// TIA Portal project "Phase_Two" (V15.1)

(* hardware
DEVICE "S71500/ET200MP-Station_1"  S7-1500 station
   slot 0: "Profilschiene_0"  6ES7 590-1***0-0AA0
   slot 1: "PLC_1"  CPU 1511-1 PN  6ES7 511-1AK00-0AB0  V1.8
   slot 2: "AI 8xU/I/RTD/TC ST_1"  AI 8xU/I/RTD/TC ST  6ES7 531-7KF00-0AB0  V2.0
   slot 3: "AI 8xU/I/RTD/TC ST_2"  AI 8xU/I/RTD/TC ST  6ES7 531-7KF00-0AB0  V2.0
   slot 4: "AI 8xU/I/RTD/TC ST_3"  AI 8xU/I/RTD/TC ST  6ES7 531-7KF00-0AB0  V2.0
   slot 5: "AI 8xU/I/RTD/TC ST_4"  AI 8xU/I/RTD/TC ST  6ES7 531-7KF00-0AB0  V2.0
   slot 6: "DI 16x24VDC BA_1"  DI 16x24VDC BA  6ES7 521-1BH10-0AA0  V1.0
   slot 7: "AI 8xU/I/RTD/TC ST_5"  AI 8xU/I/RTD/TC ST  6ES7 531-7KF00-0AB0  V2.0
DEVICE "HMI_2"  TP1200 Comfort
   slot 0: "HMI_2"  TP1200 Comfort  6AV2 124-0MC01-0AX0  15.1.0.0
   slot 1: "HMI_RT_2"  TP1200 Comfort  6AV2 124-0MC01-0AX0  15.1.0.0
   slot 5: "HMI_2.IE_CP_1"  PROFINET Interface  15.0.1.0
      slot 1: "PROFINET Interface_1"  PROFINET Interface
         slot 1: "Port_1"  Port
         slot 2: "Port_2"  Port
   slot 7: "HMI_2.MPI/DP_CP_1"  MPI/DP Interface  15.0.1.0
*)

// ===== PLC "PLC_1"  CPU 1511-1 PN =====

VAR_GLOBAL   // PLC tag table "Standard-Variablentabelle"
   "Item at entry" AT %E0.0 : Bool;
   "Item at Exit" AT %I0.1 : Bool;
   "Moving x" AT %I0.2 : Bool;
   "Item Detected" AT %I0.4 : Bool;
   "Start" AT %I0.5 : Bool;
   "Reset" AT %I0.6 : Bool;
   "Stop" AT %I0.7 : Bool;
   "Entry Conveyor" AT %QW6 : Word;
   "Exit Conveyor" AT %QW8 : Word;
   "Move x" AT %QW18 : Word;
   "Move z" AT %QW20 : Word;
   "Grab" AT %Q0.4 : Bool;
   "Start Light" AT %Q0.5 : Bool;
   "Reset Light" AT %Q0.6 : Bool;
   "Stop Light" AT %Q0.7 : Bool;
   "Moving Z" AT %I0.3 : Bool;
   "-ve edge z" AT %M7.0 : Bool;
   "Emergency Stop" AT %I1.0 : Bool;
   "-ve edge x" AT %M7.1 : Bool;
   "-ve edge to start z" AT %M7.2 : Bool;
   "-ve edge to start x" AT %M7.3 : Bool;
   "o/ps off" AT %M7.4 : Bool;
   "stop tag" AT %M7.5 : Bool;
   "Entry_conv_true" AT %M0.0 : Bool;
   "Norm_Entry_conv" AT %MD100 : Real;
   "Exit_Conv_true" AT %M0.1 : Bool;
   "Norm_Exit_conv" AT %MD104 : Real;
   "Feeding_Curved_Conv" AT %QW10 : Word;
   "Norm_Feeding_Curved_Conv" AT %MD108 : Real;
   "To Sorting Conv" AT %QW12 : Word;
   "Blue Conv" AT %QW14 : Word;
   "Green Conv" AT %QW16 : Word;
   "Sorting Rollers" AT %Q1.0 : Bool;
   "Right Pose" AT %Q1.1 : Bool;
   "Left Pose" AT %Q1.2 : Bool;
   "Vision Sensor Blue" AT %I1.3 : Bool;
   "Vision Sensor Green" AT %I1.4 : Bool;
   "Move_x_True" AT %M0.2 : Bool;
   "Move_z_True" AT %M0.3 : Bool;
   "Moving_x_Normalized" AT %M0.4 : Bool;
   "Moving_z_Normalized" AT %M0.5 : Bool;
   "Norm_Move_x" AT %MD112 : Real;
   "Norm _Move z" AT %MD116 : Real;
   "Start Green Conv sesnor" AT %I1.5 : Bool;
   "Start Blue Conv sensor" AT %I1.6 : Bool;
   "Start Green conv bit" AT %M0.6 : Bool;
   "Start Blue Conv bit" AT %M0.7 : Bool;
   "Green Machining Sensor Exit" AT %I2.0 : Bool;
   "Blue Machining Sensor Exit" AT %I1.7 : Bool;
   "Blue Conv 2" AT %QW22 : Word;
   "Green Conv 2" AT %QW24 : Word;
   "Green Conv 3" AT %QW26 : Word;
   "Green Conv 4" AT %QW28 : Word;
   "Machining Blue Start" AT %Q1.3 : Bool;
   "Machining Blue prod_lid" AT %Q1.4 : Bool;
   "-ve edge to start b_machining" AT %M10.0 : Bool;
   "Start b_machining bit" AT %M10.1 : Bool;
   "-ve edge to start g_machining" AT %M10.2 : Bool;
   "Start g_machining bit" AT %M10.3 : Bool;
   "Machining Green Start" AT %Q1.5 : Bool;
   "Machining Green prod_lid" AT %Q1.6 : Bool;
   "Green Conv after mach." AT %QW30 : Word;
   "Blue Conv after mach." AT %QW32 : Word;
   "Green Conv to Assembly" AT %QW34 : Word;
   "Curvred Green Conv assembly" AT %QW36 : Word;
   "Green lid Conv Assembly" AT %QW38 : Word;
   "Green Base Conv Assembly" AT %QW40 : Word;
   "Move_x Green Asssembly" AT %QW42 : Word;
   "Move_z Green Assembly" AT %QW44 : Word;
   "Moving_x Green Assembly" AT %I2.1 : Bool;
   "Moving_z Green Assembly" AT %I2.2 : Bool;
   "Item Detected Green Assembly" AT %I2.3 : Bool;
   "Grab Green Assembly" AT %Q1.7 : Bool;
   "Green Base Assembly Sensor" AT %I2.4 : Bool;
   "Green Lid Assembly Sensor" AT %I2.5 : Bool;
   "Green Base Vision Sensor" AT %I2.6 : Bool;
   "Pusher Green Base" AT %Q2.0 : Bool;
   "Pusher Green F_Limit" AT %I2.7 : Bool;
   "+ve edge Pusher Green" AT %M12.0 : Bool;
   "+ve edge Pusher Green true" AT %M12.1 : Bool;
   "Green Lid Vision Sensor" AT %I3.0 : Bool;
   "+ve edge green base sesnsor" AT %M15.0 : Bool;
   "+ve edge green lid sensor" AT %M15.1 : Bool;
   "Clamp Green Lid" AT %Q2.1 : Bool;
   "Clamp Green Base" AT %Q2.2 : Bool;
   "Green Base Clamped" AT %I3.2 : Bool;
   "Green Lid Clamped" AT %I3.1 : Bool;
   "Green Product Raise" AT %Q2.3 : Bool;
   "Green Product Base Limit" AT %I3.3 : Bool;
   "+ve edge to release clamp ( Green base)" AT %M20.0 : Bool;
   "+ve edge to release G Base true" AT %M20.1 : Bool;
   "Tag_1" AT %M50.0 : Bool;
   "Tag_2" AT %M25.0 : Bool;
   "Tag_3" AT %M60.0 : Bool;
   "Tag_4" AT %M61.0 : Bool;
   "+ve edge to release G lid (true)" AT %M61.1 : Bool;
   "Tag_5" AT %M65.0 : Bool;
   "Tag_6" AT %M80.0 : Bool;
   "Move z True green" AT %M80.1 : Bool;
   "move x True green" AT %M80.2 : Bool;
   "Tag_7" AT %M30.0 : Bool;
   "Tag_8" AT %M30.1 : Bool;
   "-ve edge to start x green" AT %M30.2 : Bool;
   "Move_x Green True" AT %M30.3 : Bool;
   "Tag_9" AT %M150.0 : Bool;
   "-ve edge to start z green" AT %M150.1 : Bool;
   "o/ps off green" AT %M200.0 : Bool;
   "Tag_10" AT %M210.0 : Bool;
   "Tag_11" AT %M55.0 : Bool;
   "FreeBase" AT %M30.4 : Bool;
   "Tag_12" AT %M40.0 : Bool;
   "Tag_13" AT %M40.1 : Bool;
   "Tag_14" AT %M40.3 : Bool;
   "Tag_15" AT %M40.2 : Bool;
   "Tag_16" AT %M40.4 : Bool;
   "Tag_17" AT %M40.5 : Bool;
   "Tag_18" AT %M40.6 : Bool;
   "Tag_19" AT %M40.7 : Bool;
   "Tag_20" AT %M41.0 : Bool;
   "GreenPositionerRaise" AT %Q2.4 : Bool;
   "Tag_21" AT %M41.2 : Bool;
   "Tag_22" AT %M41.3 : Bool;
   "Tag_23" AT %M41.4 : Bool;
   "Tag_24" AT %M41.5 : Bool;
   "Tag_25" AT %M41.6 : Bool;
   "Blue Base Assembly Sensor" AT %I3.7 : Bool;
   "Blue Lid Assembly Sensor" AT %I4.0 : Bool;
   "Blue Base Clamped" AT %I4.1 : Bool;
   "Blue Lid Clamped" AT %I4.2 : Bool;
   "Blue Product Counter Sensor" AT %I4.3 : Bool;
   "Blue Pusher Front Limit" AT %I4.4 : Bool;
   "Item Detected Blue" AT %I3.6 : Bool;
   "Grab Blue" AT %Q2.5 : Bool;
   "Blue Base Clamp" AT %Q2.6 : Bool;
   "Blue lid Clamp" AT %Q2.7 : Bool;
   "Blue Base Freed" AT %Q3.0 : Bool;
   "Blue lid Freed" AT %Q3.1 : Bool;
   "Pusher Blue Base" AT %Q3.2 : Bool;
   "Vision Sensor Blue base" AT %IW5 : Word;
   "Move_X Blue" AT %QW46 : Word;
   "Move_Z Blue" AT %QW48 : Word;
   "Blue Base Conv Assembly" AT %QW50 : Word;
   "Curved Blue Lid Conv Assembly" AT %QW52 : Word;
   "Blue Lid Conv Assembly" AT %QW54 : Word;
   "Moving_X Blue" AT %I4.5 : Bool;
   "Moving_Z Blue" AT %I4.6 : Bool;
   "Blue Base sensor" AT %M300.0 : Bool;
   "+ve edge Pusher blue true" AT %M300.1 : Bool;
   "Tag_26" AT %M300.2 : Bool;
   "Tag_27" AT %M300.3 : Bool;
   "Blue Lid Sensor" AT %M300.4 : Bool;
   "Tag_28" AT %M300.5 : Bool;
   "Tag_29" AT %M300.6 : Bool;
   "Tag_30" AT %M300.7 : Bool;
   "-ve edge to start Z blue" AT %M301.0 : Bool;
   "Free base blue" AT %M301.1 : Bool;
   "Tag_31" AT %M301.2 : Bool;
   "Tag_32" AT %M301.3 : Bool;
   "+ve edge to relase  b lid (true)" AT %M301.4 : Bool;
   "Tag_33" AT %M301.5 : Bool;
   "Tag_34" AT %M301.6 : Bool;
   "Move z true Blue" AT %M301.7 : Bool;
   "Tag_35" AT %M302.0 : Bool;
   "Tag_36" AT %M5.0 : Bool;
   "Tag_37" AT %M302.2 : Bool;
   "Tag_38" AT %M500.1 : Bool;
   "Tag_39" AT %M302.4 : Bool;
   "-ve edge to start X blue" AT %M302.5 : Bool;
   "Tag_40" AT %M302.6 : Bool;
   "Move_x Blue True" AT %M302.7 : Bool;
   "Tag_41" AT %M303.0 : Bool;
   "Tag_42" AT %M303.1 : Bool;
   "Tag_43" AT %M303.2 : Bool;
   "Blue Product Base Limit" AT %I3.5 : Bool;
   "Tag_44" AT %M303.4 : Bool;
   "Tag_45" AT %M303.5 : Bool;
   "Tag_46" AT %M303.6 : Bool;
   "Tag_47" AT %M303.7 : Bool;
   "Tag_48" AT %M304.0 : Bool;
   "Tag_49" AT %M304.1 : Bool;
   "Tag_50" AT %M500.2 : Bool;
   "Tag_51" AT %M600.0 : Bool;
   "tag_52" AT %M600.1 : Bool;
   "Tag_53" AT %M600.2 : Bool;
   "Tag_54" AT %M600.3 : Bool;
   "RequiredGreen" AT %MW700 : Word;
   "RequiredBlue" AT %MW702 : Word;
   "DoubleRequiredBlue" AT %MW704 : Word;
   "DoubleRequiredGreen" AT %MW706 : Word;
   "ReachedBlueItems" AT %M600.4 : Bool;
   "ReachedGreenItems" AT %M600.5 : Bool;
   "GreenProductCounterSensor" AT %I3.4 : Bool;
   "DoneGreen" AT %MW708 : Word;
   "DoneBlue" AT %MW710 : Word;
   "RequiredBlue+1" AT %MW712 : Word;
   "RequiredGreen+1" AT %MW714 : Word;
   "Reset_Tag" AT %M600.6 : Bool;
   "DoubleRequiredBlue+1" AT %MW716 : Word;
   "DoubleRequiredGreen+1" AT %MW718 : Word;
   "InputConvOFF" AT %M600.7 : Bool;
   "ReachedRawGreen" AT %M601.0 : Bool;
   "ReachedRawBlue" AT %M601.1 : Bool;
   "ConvSpeedBeforeMach" AT %MW720 : Word;
   "ConvSpeedAfterMach" AT %MW722 : Word;
   "StopConvBM" AT %M601.2 : Bool;
   "Reset_Tag_2" AT %M601.3 : Bool;
   "StartFromHmi" AT %M601.4 : Bool;
   "StopFromHmi" AT %M601.5 : Bool;
   "ResetFromHmi" AT %M601.6 : Bool;
   "Conv_Speed_Before_mach_Hmi" AT %MW724 : Word;
   "Conv_Speed_after_mach_Hmi" AT %MW726 : Word;
   "Normalized Conv Before mach" AT %MD120 : Real;
   "Normalized Conv After mach" AT %MD124 : Real;
END_VAR

// folder: System blocks/Program resources

DATA_BLOCK "IEC_Timer_0_DB"   // DB1
{ S7_Optimized_Access := 'TRUE' }
AUTHOR : Simatic
FAMILY : IEC
NAME : IEC_TMR
VERSION : 1.0
// stored: InstanceOfName IEC_TIMER
"IEC_TIMER"
BEGIN
END_DATA_BLOCK

DATA_BLOCK "IEC_Counter_0_DB"   // DB3
{ S7_Optimized_Access := 'TRUE' }
AUTHOR : Simatic
FAMILY : IEC
NAME : CNTR
VERSION : 1.0
// stored: InstanceOfName IEC_COUNTER
"IEC_COUNTER"
BEGIN
END_DATA_BLOCK

DATA_BLOCK "IEC_Counter_0_DB_1"   // DB4
{ S7_Optimized_Access := 'TRUE' }
AUTHOR : Simatic
FAMILY : IEC
NAME : CNTR
VERSION : 1.0
// stored: InstanceOfName IEC_COUNTER
"IEC_COUNTER"
BEGIN
END_DATA_BLOCK

DATA_BLOCK "IEC_Counter_0_DB_2"   // DB5
{ S7_Optimized_Access := 'TRUE' }
AUTHOR : Simatic
FAMILY : IEC
NAME : CNTR
VERSION : 1.0
// stored: InstanceOfName IEC_COUNTER
"IEC_COUNTER"
BEGIN
END_DATA_BLOCK

DATA_BLOCK "IEC_Counter_0_DB_3"   // DB6
{ S7_Optimized_Access := 'TRUE' }
AUTHOR : Simatic
FAMILY : IEC
NAME : CNTR
VERSION : 1.0
// stored: InstanceOfName IEC_COUNTER
"IEC_COUNTER"
BEGIN
END_DATA_BLOCK

DATA_BLOCK "IEC_Counter_0_DB_4"   // DB7
{ S7_Optimized_Access := 'TRUE' }
AUTHOR : Simatic
FAMILY : IEC
NAME : CNTR
VERSION : 1.0
// stored: InstanceOfName IEC_COUNTER
"IEC_COUNTER"
BEGIN
END_DATA_BLOCK

DATA_BLOCK "IEC_Timer_0_DB_4"   // DB8
{ S7_Optimized_Access := 'TRUE' }
AUTHOR : Simatic
FAMILY : IEC
NAME : IEC_TMR
VERSION : 1.0
// stored: InstanceOfName IEC_TIMER
"IEC_TIMER"
BEGIN
END_DATA_BLOCK

DATA_BLOCK "IEC_Timer_0_DB_5"   // DB9
{ S7_Optimized_Access := 'TRUE' }
AUTHOR : Simatic
FAMILY : IEC
NAME : IEC_TMR
VERSION : 1.0
// stored: InstanceOfName IEC_TIMER
"IEC_TIMER"
BEGIN
END_DATA_BLOCK

DATA_BLOCK "IEC_Timer_0_DB_6"   // DB10
{ S7_Optimized_Access := 'TRUE' }
AUTHOR : Simatic
FAMILY : IEC
NAME : IEC_TMR
VERSION : 1.0
// stored: InstanceOfName IEC_TIMER
"IEC_TIMER"
BEGIN
END_DATA_BLOCK

DATA_BLOCK "IEC_Timer_0_DB_7"   // DB11
{ S7_Optimized_Access := 'TRUE' }
AUTHOR : Simatic
FAMILY : IEC
NAME : IEC_TMR
VERSION : 1.0
// stored: InstanceOfName IEC_TIMER
"IEC_TIMER"
BEGIN
END_DATA_BLOCK

DATA_BLOCK "IEC_Counter_0_DB_5"   // DB12
{ S7_Optimized_Access := 'TRUE' }
AUTHOR : Simatic
FAMILY : IEC
NAME : CNTR
VERSION : 1.0
// stored: InstanceOfName IEC_COUNTER
"IEC_COUNTER"
BEGIN
END_DATA_BLOCK

DATA_BLOCK "IEC_Counter_0_DB_6"   // DB13
{ S7_Optimized_Access := 'TRUE' }
AUTHOR : Simatic
FAMILY : IEC
NAME : CNTR
VERSION : 1.0
// stored: InstanceOfName IEC_COUNTER
"IEC_COUNTER"
BEGIN
END_DATA_BLOCK

DATA_BLOCK "IEC_Timer_0_DB_2"   // DB14
{ S7_Optimized_Access := 'TRUE' }
AUTHOR : Simatic
FAMILY : IEC
NAME : IEC_TMR
VERSION : 1.0
// stored: InstanceOfName IEC_TIMER
"IEC_TIMER"
BEGIN
END_DATA_BLOCK

DATA_BLOCK "IEC_Timer_0_DB_3"   // DB15
{ S7_Optimized_Access := 'TRUE' }
AUTHOR : Simatic
FAMILY : IEC
NAME : IEC_TMR
VERSION : 1.0
// stored: InstanceOfName IEC_TIMER
"IEC_TIMER"
BEGIN
END_DATA_BLOCK

// folder: (top level)

FUNCTION "MHJ-PLC-Lab-Function-S71500" : Void   // FC9000, SCL
{ S7_Optimized_Access := 'TRUE' }
VERSION : 0.1
   VAR_TEMP
      Value : Byte;
      ForCounter : Int;
   END_VAR
   VAR CONSTANT
      Value_01_DW : DWord := 16#1223_5486;
      Value_02_DW : DWord := 16#A6C9_D1F5;
   END_VAR
BEGIN

   #Value:=PEEK(area := 16#82,
        dbNumber := 0,
        byteOffset := 511);
   #Value := #Value + 1;

   POKE(area := 16#82,
        dbNumber := 0,
        byteOffset := 511,
        value := #Value);

   POKE(area := 16#82,
        dbNumber := 0,
        byteOffset := 1016,
        value := #Value_01_DW);
   POKE(area := 16#82,
        dbNumber := 0,
        byteOffset := 1020,
        value := #Value_02_DW);

   FOR #ForCounter := 0 TO 63 DO
       #Value:=PEEK(area := 16#1,
            dbNumber := 0,
            byteOffset := #ForCounter);
       POKE(area := 16#81,
            dbNumber := 0,
            byteOffset := #ForCounter,
            value := #Value);
   END_FOR;
   #Value := PEEK(area := 16#1,
                  dbNumber := 0,
                  byteOffset := 512);
   POKE(area := 16#82,
        dbNumber := 0,
        byteOffset := 512,
        value := #Value);
END_FUNCTION

ORGANIZATION_BLOCK "Main"   // OB1, FBD, ProgramCycle
TITLE = "Main Program Sweep (Cycle)"
{ S7_Optimized_Access := 'TRUE' }
VERSION : 0.1
   VAR_INPUT
      Initial_Call : Bool;   // Initial call of this OB
      Remanence : Bool;   // =True, if remanent data are available
   END_VAR
BEGIN

REGION Network 1
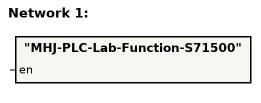
   "MHJ-PLC-Lab-Function-S71500"();
END_REGION
END_ORGANIZATION_BLOCK

ORGANIZATION_BLOCK "Main_1"   // OB123, LAD, ProgramCycle
TITLE = "Main Program Sweep (Cycle)"
{ S7_Optimized_Access := 'TRUE' }
VERSION : 0.1
   VAR_INPUT
      Initial_Call : Bool;   // Initial call of this OB
      Remanence : Bool;   // =True, if remanent data are available
   END_VAR
   VAR_TEMP   // added for the SCL form of the ladder/FBD networks
      _w1 : Bool;
      _w2 : Bool;
      _w3 : Bool;
      _w4 : Bool;
   END_VAR
BEGIN

REGION Network 1
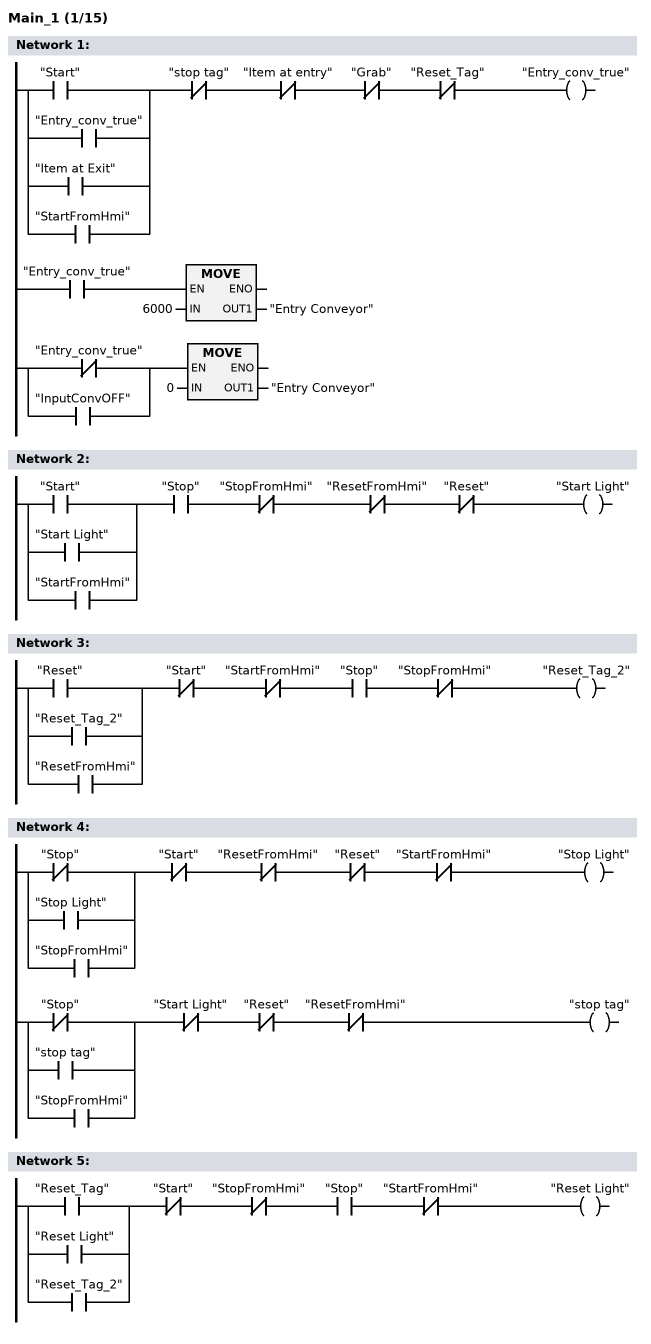
   RUNG wire#powerrail
      Contact( "Start" )
      wire#w1
      I_Contact( "stop tag" )
      I_Contact( "Item at entry" )
      I_Contact( "Grab" )
      I_Contact( "Reset_Tag" )
      Coil( "Entry_conv_true" )
   END_RUNG
   RUNG wire#powerrail
      Contact( "Entry_conv_true" )
   END_RUNG wire#w1
   RUNG wire#powerrail
      Contact( "Item at Exit" )
   END_RUNG wire#w1
   RUNG wire#powerrail
      Contact( "StartFromHmi" )
   END_RUNG wire#w1
   RUNG wire#powerrail
      Contact( "Entry_conv_true" )
      Move(in := 6000, out1 => "Entry Conveyor")
   END_RUNG
   RUNG wire#powerrail
      I_Contact( "Entry_conv_true" )
      wire#w2
      Move(in := 0, out1 => "Entry Conveyor")
   END_RUNG
   RUNG wire#powerrail
      Contact( "InputConvOFF" )
   END_RUNG wire#w2
   // the same network as SCL:
   "Entry_conv_true" := ("Start" OR "Entry_conv_true" OR "Item at Exit" OR "StartFromHmi") AND NOT "stop tag" AND NOT "Item at entry" AND NOT "Grab" AND NOT "Reset_Tag";
   IF "Entry_conv_true" THEN "Entry Conveyor" := 6000; END_IF;
   IF NOT "Entry_conv_true" OR "InputConvOFF" THEN "Entry Conveyor" := 0; END_IF;
END_REGION

REGION Network 2
   RUNG wire#powerrail
      Contact( "Start" )
      wire#w1
      Contact( "Stop" )
      I_Contact( "StopFromHmi" )
      I_Contact( "ResetFromHmi" )
      I_Contact( "Reset" )
      Coil( "Start Light" )
   END_RUNG
   RUNG wire#powerrail
      Contact( "Start Light" )
   END_RUNG wire#w1
   RUNG wire#powerrail
      Contact( "StartFromHmi" )
   END_RUNG wire#w1
   // the same network as SCL:
   "Start Light" := ("Start" OR "Start Light" OR "StartFromHmi") AND "Stop" AND NOT "StopFromHmi" AND NOT "ResetFromHmi" AND NOT "Reset";
END_REGION

REGION Network 3
   RUNG wire#powerrail
      Contact( "Reset" )
      wire#w1
      I_Contact( "Start" )
      I_Contact( "StartFromHmi" )
      Contact( "Stop" )
      I_Contact( "StopFromHmi" )
      Coil( "Reset_Tag_2" )
   END_RUNG
   RUNG wire#powerrail
      Contact( "Reset_Tag_2" )
   END_RUNG wire#w1
   RUNG wire#powerrail
      Contact( "ResetFromHmi" )
   END_RUNG wire#w1
   // the same network as SCL:
   "Reset_Tag_2" := ("Reset" OR "Reset_Tag_2" OR "ResetFromHmi") AND NOT "Start" AND NOT "StartFromHmi" AND "Stop" AND NOT "StopFromHmi";
END_REGION

REGION Network 4
   RUNG wire#powerrail
      I_Contact( "Stop" )
      wire#w1
      I_Contact( "Start" )
      I_Contact( "ResetFromHmi" )
      I_Contact( "Reset" )
      I_Contact( "StartFromHmi" )
      Coil( "Stop Light" )
   END_RUNG
   RUNG wire#powerrail
      Contact( "Stop Light" )
   END_RUNG wire#w1
   RUNG wire#powerrail
      Contact( "StopFromHmi" )
   END_RUNG wire#w1
   RUNG wire#powerrail
      I_Contact( "Stop" )
      wire#w2
      I_Contact( "Start Light" )
      I_Contact( "Reset" )
      I_Contact( "ResetFromHmi" )
      Coil( "stop tag" )
   END_RUNG
   RUNG wire#powerrail
      Contact( "stop tag" )
   END_RUNG wire#w2
   RUNG wire#powerrail
      Contact( "StopFromHmi" )
   END_RUNG wire#w2
   // the same network as SCL:
   "Stop Light" := (NOT "Stop" OR "Stop Light" OR "StopFromHmi") AND NOT "Start" AND NOT "ResetFromHmi" AND NOT "Reset" AND NOT "StartFromHmi";
   "stop tag" := (NOT "Stop" OR "stop tag" OR "StopFromHmi") AND NOT "Start Light" AND NOT "Reset" AND NOT "ResetFromHmi";
END_REGION

REGION Network 5
   RUNG wire#powerrail
      Contact( "Reset_Tag" )
      wire#w1
      I_Contact( "Start" )
      I_Contact( "StopFromHmi" )
      Contact( "Stop" )
      I_Contact( "StartFromHmi" )
      Coil( "Reset Light" )
   END_RUNG
   RUNG wire#powerrail
      Contact( "Reset Light" )
   END_RUNG wire#w1
   RUNG wire#powerrail
      Contact( "Reset_Tag_2" )
   END_RUNG wire#w1
   // the same network as SCL:
   "Reset Light" := ("Reset_Tag" OR "Reset Light" OR "Reset_Tag_2") AND NOT "Start" AND NOT "StopFromHmi" AND "Stop" AND NOT "StartFromHmi";
END_REGION

REGION Network 6
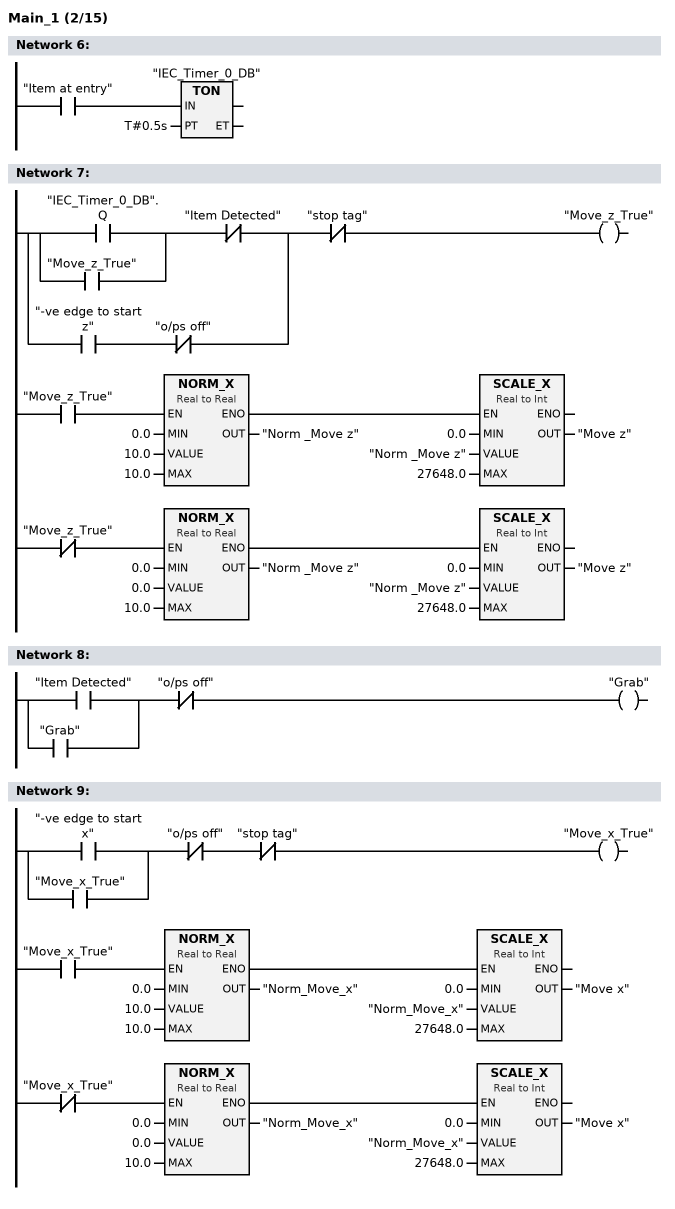
   "IEC_Timer_0_DB".TON(IN := "Item at entry", PT := T#0.5s);
END_REGION

REGION Network 7
   RUNG wire#powerrail
      Contact( "IEC_Timer_0_DB".Q )
      wire#w1
      I_Contact( "Item Detected" )
      wire#w2
      I_Contact( "stop tag" )
      Coil( "Move_z_True" )
   END_RUNG
   RUNG wire#powerrail
      Contact( "Move_z_True" )
   END_RUNG wire#w1
   RUNG wire#powerrail
      Contact( "-ve edge to start z" )
      I_Contact( "o/ps off" )
   END_RUNG wire#w2
   RUNG wire#powerrail
      Contact( "Move_z_True" )
      { S7_Templates := "[SrcType := Real, DestType := Real]" } Normalize(min := 0.0, value := 10.0, max := 10.0, out => "Norm _Move z")
      { S7_Templates := "[SrcType := Real, DestType := Int]" } Scale(min := 0.0, value := "Norm _Move z", max := 27648.0, out => "Move z")
   END_RUNG
   RUNG wire#powerrail
      I_Contact( "Move_z_True" )
      { S7_Templates := "[SrcType := Real, DestType := Real]" } Normalize(min := 0.0, value := 0.0, max := 10.0, out => "Norm _Move z")
      { S7_Templates := "[SrcType := Real, DestType := Int]" } Scale(min := 0.0, value := "Norm _Move z", max := 27648.0, out => "Move z")
   END_RUNG
   // the same network as SCL:
   "Move_z_True" := ((("IEC_Timer_0_DB".Q OR "Move_z_True") AND NOT "Item Detected") OR ("-ve edge to start z" AND NOT "o/ps off")) AND NOT "stop tag";
   IF "Move_z_True" THEN
       "Norm _Move z" := NORM_X(MIN := 0.0, VALUE := 10.0, MAX := 10.0);
       "Move z" := SCALE_X(MIN := 0.0, VALUE := "Norm _Move z", MAX := 27648.0);
   END_IF;
   IF NOT "Move_z_True" THEN
       "Norm _Move z" := NORM_X(MIN := 0.0, VALUE := 0.0, MAX := 10.0);
       "Move z" := SCALE_X(MIN := 0.0, VALUE := "Norm _Move z", MAX := 27648.0);
   END_IF;
END_REGION

REGION Network 8
   RUNG wire#powerrail
      Contact( "Item Detected" )
      wire#w1
      I_Contact( "o/ps off" )
      Coil( "Grab" )
   END_RUNG
   RUNG wire#powerrail
      Contact( "Grab" )
   END_RUNG wire#w1
   // the same network as SCL:
   "Grab" := ("Item Detected" OR "Grab") AND NOT "o/ps off";
END_REGION

REGION Network 9
   RUNG wire#powerrail
      Contact( "-ve edge to start x" )
      wire#w1
      I_Contact( "o/ps off" )
      I_Contact( "stop tag" )
      Coil( "Move_x_True" )
   END_RUNG
   RUNG wire#powerrail
      Contact( "Move_x_True" )
   END_RUNG wire#w1
   RUNG wire#powerrail
      Contact( "Move_x_True" )
      { S7_Templates := "[SrcType := Real, DestType := Real]" } Normalize(min := 0.0, value := 10.0, max := 10.0, out => "Norm_Move_x")
      { S7_Templates := "[SrcType := Real, DestType := Int]" } Scale(min := 0.0, value := "Norm_Move_x", max := 27648.0, out => "Move x")
   END_RUNG
   RUNG wire#powerrail
      I_Contact( "Move_x_True" )
      { S7_Templates := "[SrcType := Real, DestType := Real]" } Normalize(min := 0.0, value := 0.0, max := 10.0, out => "Norm_Move_x")
      { S7_Templates := "[SrcType := Real, DestType := Int]" } Scale(min := 0.0, value := "Norm_Move_x", max := 27648.0, out => "Move x")
   END_RUNG
   // the same network as SCL:
   "Move_x_True" := ("-ve edge to start x" OR "Move_x_True") AND NOT "o/ps off" AND NOT "stop tag";
   IF "Move_x_True" THEN
       "Norm_Move_x" := NORM_X(MIN := 0.0, VALUE := 10.0, MAX := 10.0);
       "Move x" := SCALE_X(MIN := 0.0, VALUE := "Norm_Move_x", MAX := 27648.0);
   END_IF;
   IF NOT "Move_x_True" THEN
       "Norm_Move_x" := NORM_X(MIN := 0.0, VALUE := 0.0, MAX := 10.0);
       "Move x" := SCALE_X(MIN := 0.0, VALUE := "Norm_Move_x", MAX := 27648.0);
   END_IF;
END_REGION

REGION Network 10
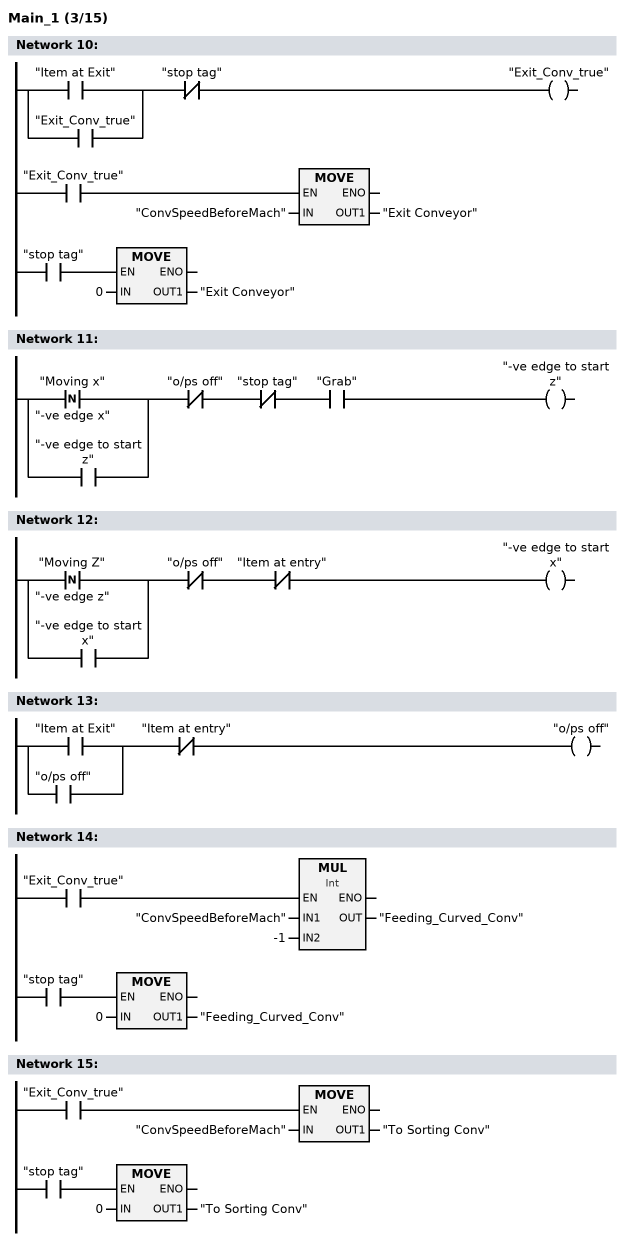
   RUNG wire#powerrail
      Contact( "Item at Exit" )
      wire#w1
      I_Contact( "stop tag" )
      Coil( "Exit_Conv_true" )
   END_RUNG
   RUNG wire#powerrail
      Contact( "Exit_Conv_true" )
   END_RUNG wire#w1
   RUNG wire#powerrail
      Contact( "Exit_Conv_true" )
      Move(in := "ConvSpeedBeforeMach", out1 => "Exit Conveyor")
   END_RUNG
   RUNG wire#powerrail
      Contact( "stop tag" )
      Move(in := 0, out1 => "Exit Conveyor")
   END_RUNG
   // the same network as SCL:
   "Exit_Conv_true" := ("Item at Exit" OR "Exit_Conv_true") AND NOT "stop tag";
   IF "Exit_Conv_true" THEN "Exit Conveyor" := "ConvSpeedBeforeMach"; END_IF;
   IF "stop tag" THEN "Exit Conveyor" := 0; END_IF;
END_REGION

REGION Network 11
   RUNG wire#powerrail
      N_Contact(operand := "Moving x", bit := "-ve edge x")
      wire#w1
      I_Contact( "o/ps off" )
      I_Contact( "stop tag" )
      Contact( "Grab" )
      Coil( "-ve edge to start z" )
   END_RUNG
   RUNG wire#powerrail
      Contact( "-ve edge to start z" )
   END_RUNG wire#w1
   // the same network as SCL:
   #_w1 := NOT "Moving x" AND "-ve edge x";   // falling edge of "Moving x"
   "-ve edge x" := "Moving x";
   "-ve edge to start z" := (#_w1 OR "-ve edge to start z") AND NOT "o/ps off" AND NOT "stop tag" AND "Grab";
END_REGION

REGION Network 12
   RUNG wire#powerrail
      N_Contact(operand := "Moving Z", bit := "-ve edge z")
      wire#w1
      I_Contact( "o/ps off" )
      I_Contact( "Item at entry" )
      Coil( "-ve edge to start x" )
   END_RUNG
   RUNG wire#powerrail
      Contact( "-ve edge to start x" )
   END_RUNG wire#w1
   // the same network as SCL:
   #_w1 := NOT "Moving Z" AND "-ve edge z";   // falling edge of "Moving Z"
   "-ve edge z" := "Moving Z";
   "-ve edge to start x" := (#_w1 OR "-ve edge to start x") AND NOT "o/ps off" AND NOT "Item at entry";
END_REGION

REGION Network 13
   RUNG wire#powerrail
      Contact( "Item at Exit" )
      wire#w1
      I_Contact( "Item at entry" )
      Coil( "o/ps off" )
   END_RUNG
   RUNG wire#powerrail
      Contact( "o/ps off" )
   END_RUNG wire#w1
   // the same network as SCL:
   "o/ps off" := ("Item at Exit" OR "o/ps off") AND NOT "Item at entry";
END_REGION

REGION Network 14
   RUNG wire#powerrail
      Contact( "Exit_Conv_true" )
      { S7_Templates := "SrcType := Int" } Mul(in1 := "ConvSpeedBeforeMach", in2 := -1, out => "Feeding_Curved_Conv")
   END_RUNG
   RUNG wire#powerrail
      Contact( "stop tag" )
      Move(in := 0, out1 => "Feeding_Curved_Conv")
   END_RUNG
   // the same network as SCL:
   IF "Exit_Conv_true" THEN "Feeding_Curved_Conv" := "ConvSpeedBeforeMach" * (-1); END_IF;
   IF "stop tag" THEN "Feeding_Curved_Conv" := 0; END_IF;
END_REGION

REGION Network 15
   RUNG wire#powerrail
      Contact( "Exit_Conv_true" )
      Move(in := "ConvSpeedBeforeMach", out1 => "To Sorting Conv")
   END_RUNG
   RUNG wire#powerrail
      Contact( "stop tag" )
      Move(in := 0, out1 => "To Sorting Conv")
   END_RUNG
   // the same network as SCL:
   IF "Exit_Conv_true" THEN "To Sorting Conv" := "ConvSpeedBeforeMach"; END_IF;
   IF "stop tag" THEN "To Sorting Conv" := 0; END_IF;
END_REGION

REGION Network 16
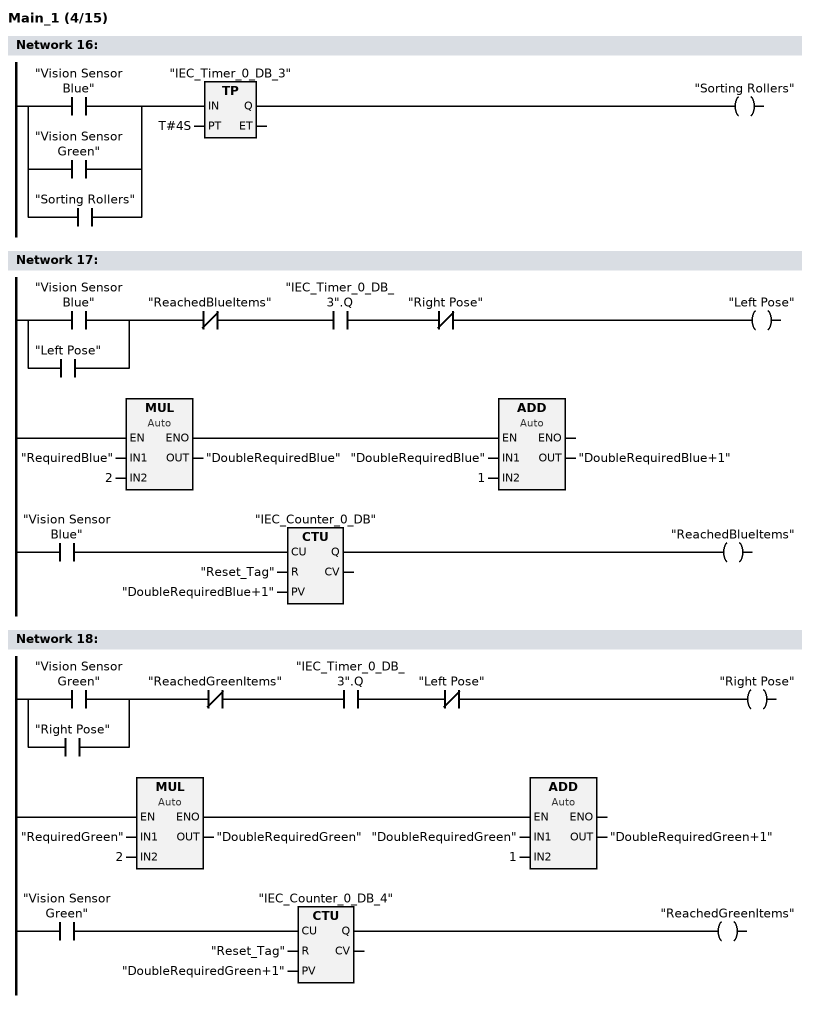
   "IEC_Timer_0_DB_3".TP(IN := "Vision Sensor Blue" OR "Vision Sensor Green" OR "Sorting Rollers", PT := T#4S);
   "Sorting Rollers" := "IEC_Timer_0_DB_3".Q;
END_REGION

REGION Network 17
   "Left Pose" := ("Vision Sensor Blue" OR "Left Pose") AND NOT "ReachedBlueItems" AND "IEC_Timer_0_DB_3".Q AND NOT "Right Pose";
   "DoubleRequiredBlue" := "RequiredBlue" * 2;
   "DoubleRequiredBlue+1" := "DoubleRequiredBlue" + 1;
   "IEC_Counter_0_DB".CTU(CU := "Vision Sensor Blue", R := "Reset_Tag", PV := "DoubleRequiredBlue+1");
   "ReachedBlueItems" := "IEC_Counter_0_DB".Q;
END_REGION

REGION Network 18
   "Right Pose" := ("Vision Sensor Green" OR "Right Pose") AND NOT "ReachedGreenItems" AND "IEC_Timer_0_DB_3".Q AND NOT "Left Pose";
   "DoubleRequiredGreen" := "RequiredGreen" * 2;
   "DoubleRequiredGreen+1" := "DoubleRequiredGreen" + 1;
   "IEC_Counter_0_DB_4".CTU(CU := "Vision Sensor Green", R := "Reset_Tag", PV := "DoubleRequiredGreen+1");
   "ReachedGreenItems" := "IEC_Counter_0_DB_4".Q;
END_REGION

REGION Network 19
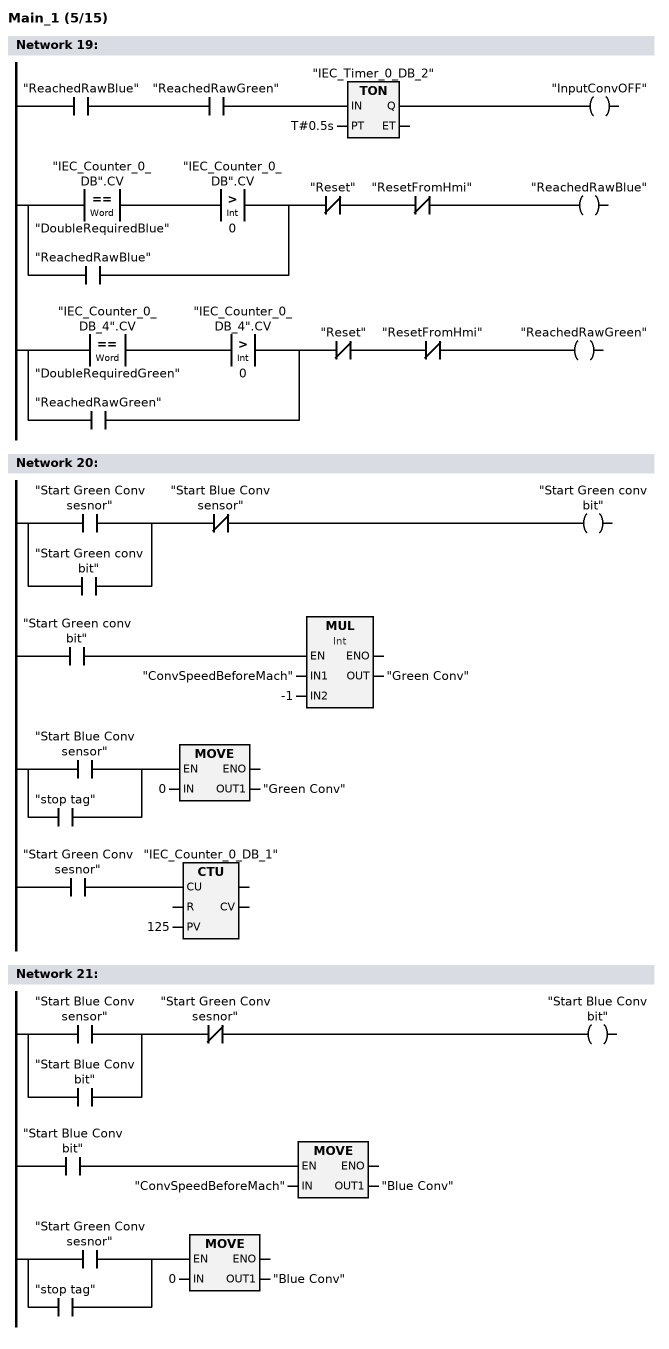
   "IEC_Timer_0_DB_2".TON(IN := "ReachedRawBlue" AND "ReachedRawGreen", PT := T#0.5s);
   "InputConvOFF" := "IEC_Timer_0_DB_2".Q;
   "ReachedRawBlue" := ((("IEC_Counter_0_DB".CV = "DoubleRequiredBlue") AND ("IEC_Counter_0_DB".CV > 0)) OR "ReachedRawBlue") AND NOT "Reset" AND NOT "ResetFromHmi";
   "ReachedRawGreen" := ((("IEC_Counter_0_DB_4".CV = "DoubleRequiredGreen") AND ("IEC_Counter_0_DB_4".CV > 0)) OR "ReachedRawGreen") AND NOT "Reset" AND NOT "ResetFromHmi";
END_REGION

REGION Network 20
   "Start Green conv bit" := ("Start Green Conv sesnor" OR "Start Green conv bit") AND NOT "Start Blue Conv sensor";
   IF "Start Green conv bit" THEN "Green Conv" := "ConvSpeedBeforeMach" * (-1); END_IF;
   IF "Start Blue Conv sensor" OR "stop tag" THEN "Green Conv" := 0; END_IF;
   "IEC_Counter_0_DB_1".CTU(CU := "Start Green Conv sesnor", PV := 125);
END_REGION

REGION Network 21
   RUNG wire#powerrail
      Contact( "Start Blue Conv sensor" )
      wire#w1
      I_Contact( "Start Green Conv sesnor" )
      Coil( "Start Blue Conv bit" )
   END_RUNG
   RUNG wire#powerrail
      Contact( "Start Blue Conv bit" )
   END_RUNG wire#w1
   RUNG wire#powerrail
      Contact( "Start Blue Conv bit" )
      Move(in := "ConvSpeedBeforeMach", out1 => "Blue Conv")
   END_RUNG
   RUNG wire#powerrail
      Contact( "Start Green Conv sesnor" )
      wire#w2
      Move(in := 0, out1 => "Blue Conv")
   END_RUNG
   RUNG wire#powerrail
      Contact( "stop tag" )
   END_RUNG wire#w2
   // the same network as SCL:
   "Start Blue Conv bit" := ("Start Blue Conv sensor" OR "Start Blue Conv bit") AND NOT "Start Green Conv sesnor";
   IF "Start Blue Conv bit" THEN "Blue Conv" := "ConvSpeedBeforeMach"; END_IF;
   IF "Start Green Conv sesnor" OR "stop tag" THEN "Blue Conv" := 0; END_IF;
END_REGION

REGION Network 22
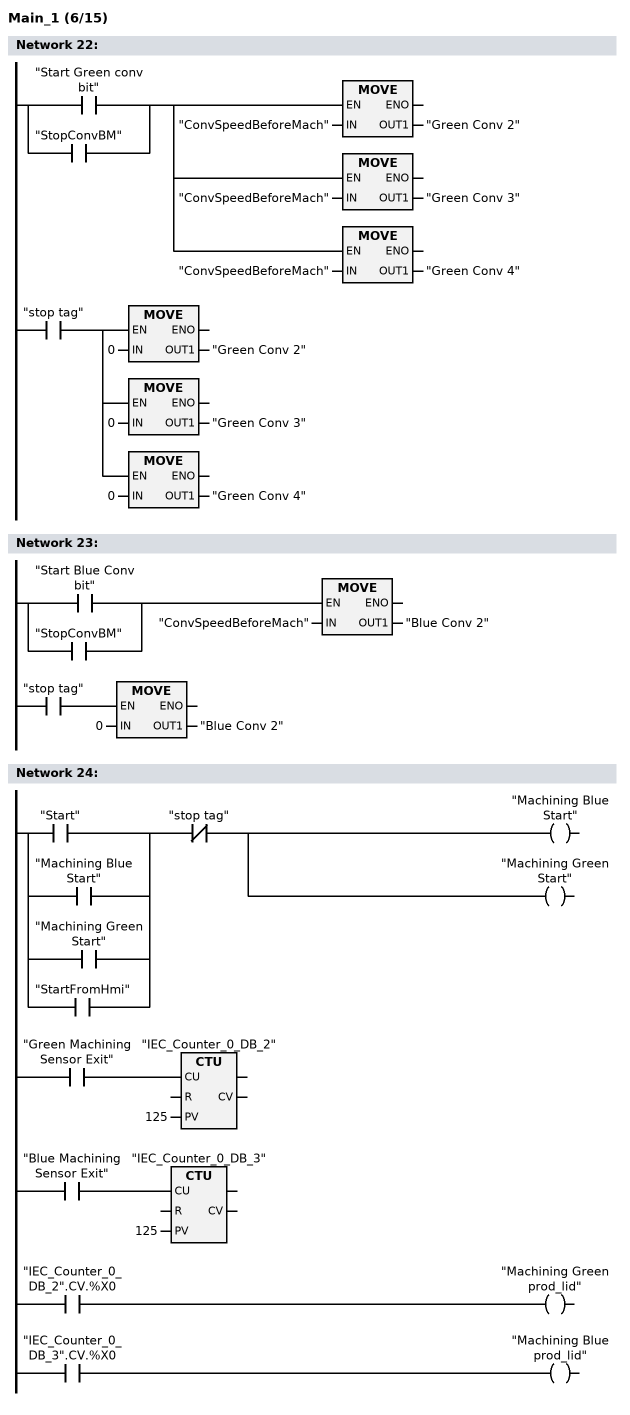
   RUNG wire#powerrail
      Contact( "Start Green conv bit" )
      wire#w1
      Move(in := "ConvSpeedBeforeMach", out1 => "Green Conv 2")
   END_RUNG
   RUNG wire#powerrail
      Contact( "StopConvBM" )
   END_RUNG wire#w1
   RUNG wire#w1
      Move(in := "ConvSpeedBeforeMach", out1 => "Green Conv 3")
   END_RUNG
   RUNG wire#w1
      Move(in := "ConvSpeedBeforeMach", out1 => "Green Conv 4")
   END_RUNG
   RUNG wire#powerrail
      Contact( "stop tag" )
      wire#w2
      Move(in := 0, out1 => "Green Conv 2")
   END_RUNG
   RUNG wire#w2
      Move(in := 0, out1 => "Green Conv 3")
   END_RUNG
   RUNG wire#w2
      Move(in := 0, out1 => "Green Conv 4")
   END_RUNG
   // the same network as SCL:
   IF "Start Green conv bit" OR "StopConvBM" THEN
       "Green Conv 2" := "ConvSpeedBeforeMach";
       "Green Conv 3" := "ConvSpeedBeforeMach";
       "Green Conv 4" := "ConvSpeedBeforeMach";
   END_IF;
   IF "stop tag" THEN
       "Green Conv 2" := 0;
       "Green Conv 3" := 0;
       "Green Conv 4" := 0;
   END_IF;
END_REGION

REGION Network 23
   RUNG wire#powerrail
      Contact( "Start Blue Conv bit" )
      wire#w1
      Move(in := "ConvSpeedBeforeMach", out1 => "Blue Conv 2")
   END_RUNG
   RUNG wire#powerrail
      Contact( "StopConvBM" )
   END_RUNG wire#w1
   RUNG wire#powerrail
      Contact( "stop tag" )
      Move(in := 0, out1 => "Blue Conv 2")
   END_RUNG
   // the same network as SCL:
   IF "Start Blue Conv bit" OR "StopConvBM" THEN "Blue Conv 2" := "ConvSpeedBeforeMach"; END_IF;
   IF "stop tag" THEN "Blue Conv 2" := 0; END_IF;
END_REGION

REGION Network 24
   "Machining Blue Start" := ("Start" OR "Machining Blue Start" OR "Machining Green Start" OR "StartFromHmi") AND NOT "stop tag";
   "Machining Green Start" := "Machining Blue Start";
   "IEC_Counter_0_DB_2".CTU(CU := "Green Machining Sensor Exit", PV := 125);
   "IEC_Counter_0_DB_3".CTU(CU := "Blue Machining Sensor Exit", PV := 125);
   "Machining Green prod_lid" := "IEC_Counter_0_DB_2".CV.%X0;
   "Machining Blue prod_lid" := "IEC_Counter_0_DB_3".CV.%X0;
END_REGION

REGION Network 25
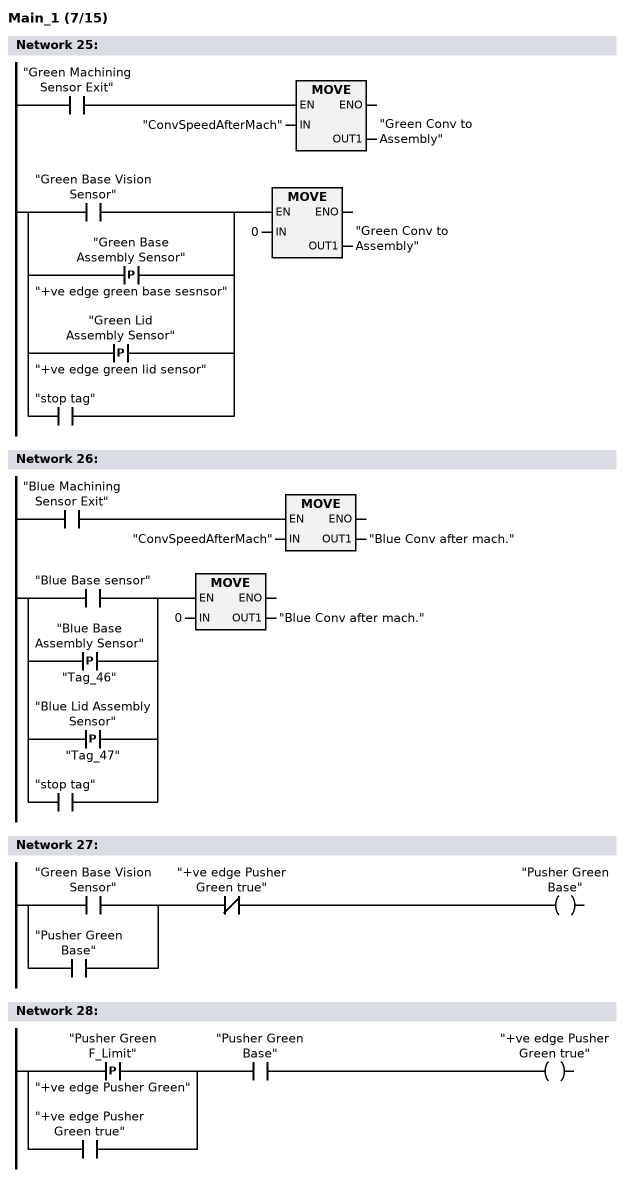
   RUNG wire#powerrail
      Contact( "Green Machining Sensor Exit" )
      Move(in := "ConvSpeedAfterMach", out1 => "Green Conv to Assembly")
   END_RUNG
   RUNG wire#powerrail
      Contact( "Green Base Vision Sensor" )
      wire#w1
      Move(in := 0, out1 => "Green Conv to Assembly")
   END_RUNG
   RUNG wire#powerrail
      P_Contact(operand := "Green Base Assembly Sensor", bit := "+ve edge green base sesnsor")
   END_RUNG wire#w1
   RUNG wire#powerrail
      P_Contact(operand := "Green Lid Assembly Sensor", bit := "+ve edge green lid sensor")
   END_RUNG wire#w1
   RUNG wire#powerrail
      Contact( "stop tag" )
   END_RUNG wire#w1
   // the same network as SCL:
   IF "Green Machining Sensor Exit" THEN "Green Conv to Assembly" := "ConvSpeedAfterMach"; END_IF;
   #_w1 := "Green Base Assembly Sensor" AND NOT "+ve edge green base sesnsor";   // rising edge of "Green Base Assembly Sensor"
   "+ve edge green base sesnsor" := "Green Base Assembly Sensor";
   #_w2 := "Green Lid Assembly Sensor" AND NOT "+ve edge green lid sensor";   // rising edge of "Green Lid Assembly Sensor"
   "+ve edge green lid sensor" := "Green Lid Assembly Sensor";
   IF "Green Base Vision Sensor" OR #_w1 OR #_w2 OR "stop tag" THEN "Green Conv to Assembly" := 0; END_IF;
END_REGION

REGION Network 26
   RUNG wire#powerrail
      Contact( "Blue Machining Sensor Exit" )
      Move(in := "ConvSpeedAfterMach", out1 => "Blue Conv after mach.")
   END_RUNG
   RUNG wire#powerrail
      Contact( "Blue Base sensor" )
      wire#w1
      Move(in := 0, out1 => "Blue Conv after mach.")
   END_RUNG
   RUNG wire#powerrail
      P_Contact(operand := "Blue Base Assembly Sensor", bit := "Tag_46")
   END_RUNG wire#w1
   RUNG wire#powerrail
      P_Contact(operand := "Blue Lid Assembly Sensor", bit := "Tag_47")
   END_RUNG wire#w1
   RUNG wire#powerrail
      Contact( "stop tag" )
   END_RUNG wire#w1
   // the same network as SCL:
   IF "Blue Machining Sensor Exit" THEN "Blue Conv after mach." := "ConvSpeedAfterMach"; END_IF;
   #_w1 := "Blue Base Assembly Sensor" AND NOT "Tag_46";   // rising edge of "Blue Base Assembly Sensor"
   "Tag_46" := "Blue Base Assembly Sensor";
   #_w2 := "Blue Lid Assembly Sensor" AND NOT "Tag_47";   // rising edge of "Blue Lid Assembly Sensor"
   "Tag_47" := "Blue Lid Assembly Sensor";
   IF "Blue Base sensor" OR #_w1 OR #_w2 OR "stop tag" THEN "Blue Conv after mach." := 0; END_IF;
END_REGION

REGION Network 27
   RUNG wire#powerrail
      Contact( "Green Base Vision Sensor" )
      wire#w1
      I_Contact( "+ve edge Pusher Green true" )
      Coil( "Pusher Green Base" )
   END_RUNG
   RUNG wire#powerrail
      Contact( "Pusher Green Base" )
   END_RUNG wire#w1
   // the same network as SCL:
   "Pusher Green Base" := ("Green Base Vision Sensor" OR "Pusher Green Base") AND NOT "+ve edge Pusher Green true";
END_REGION

REGION Network 28
   RUNG wire#powerrail
      P_Contact(operand := "Pusher Green F_Limit", bit := "+ve edge Pusher Green")
      wire#w1
      Contact( "Pusher Green Base" )
      Coil( "+ve edge Pusher Green true" )
   END_RUNG
   RUNG wire#powerrail
      Contact( "+ve edge Pusher Green true" )
   END_RUNG wire#w1
   // the same network as SCL:
   #_w1 := "Pusher Green F_Limit" AND NOT "+ve edge Pusher Green";   // rising edge of "Pusher Green F_Limit"
   "+ve edge Pusher Green" := "Pusher Green F_Limit";
   "+ve edge Pusher Green true" := (#_w1 OR "+ve edge Pusher Green true") AND "Pusher Green Base";
END_REGION

REGION Network 29
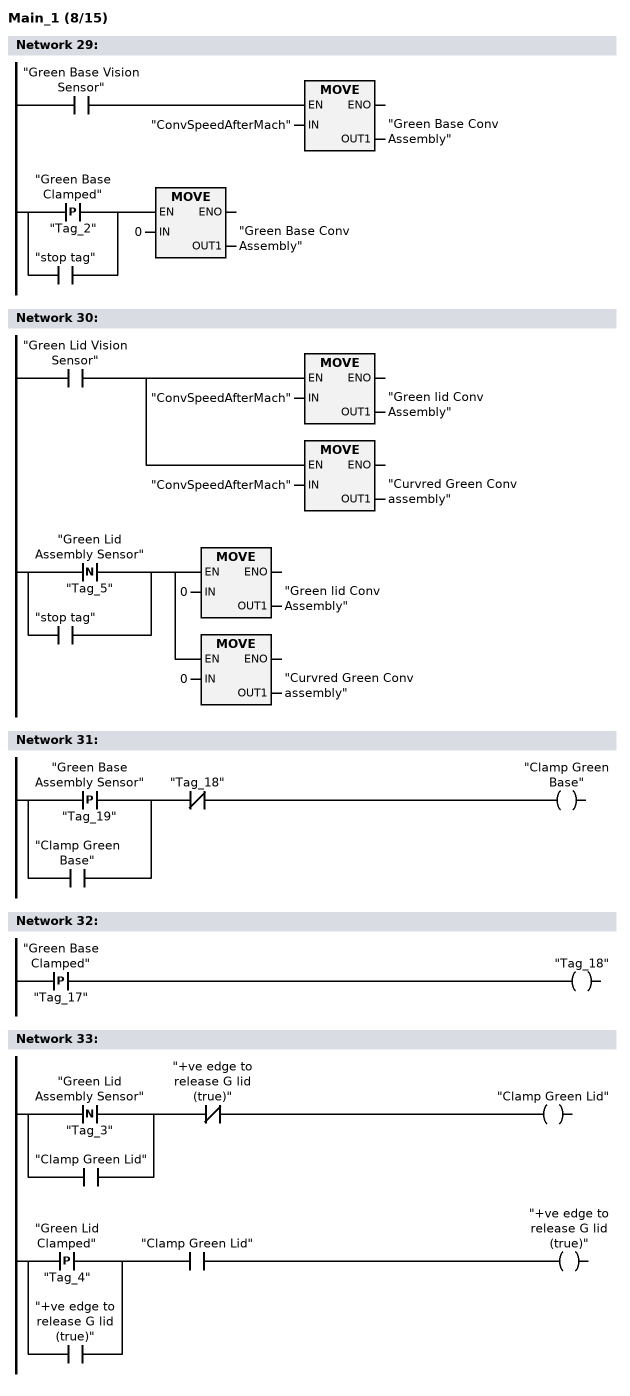
   RUNG wire#powerrail
      Contact( "Green Base Vision Sensor" )
      Move(in := "ConvSpeedAfterMach", out1 => "Green Base Conv Assembly")
   END_RUNG
   RUNG wire#powerrail
      P_Contact(operand := "Green Base Clamped", bit := "Tag_2")
      wire#w1
      Move(in := 0, out1 => "Green Base Conv Assembly")
   END_RUNG
   RUNG wire#powerrail
      Contact( "stop tag" )
   END_RUNG wire#w1
   // the same network as SCL:
   IF "Green Base Vision Sensor" THEN "Green Base Conv Assembly" := "ConvSpeedAfterMach"; END_IF;
   #_w1 := "Green Base Clamped" AND NOT "Tag_2";   // rising edge of "Green Base Clamped"
   "Tag_2" := "Green Base Clamped";
   IF #_w1 OR "stop tag" THEN "Green Base Conv Assembly" := 0; END_IF;
END_REGION

REGION Network 30
   RUNG wire#powerrail
      Contact( "Green Lid Vision Sensor" )
      wire#w1
      Move(in := "ConvSpeedAfterMach", out1 => "Green lid Conv Assembly")
   END_RUNG
   RUNG wire#w1
      Move(in := "ConvSpeedAfterMach", out1 => "Curvred Green Conv assembly")
   END_RUNG
   RUNG wire#powerrail
      N_Contact(operand := "Green Lid Assembly Sensor", bit := "Tag_5")
      wire#w2
      Move(in := 0, out1 => "Green lid Conv Assembly")
   END_RUNG
   RUNG wire#powerrail
      Contact( "stop tag" )
   END_RUNG wire#w2
   RUNG wire#w2
      Move(in := 0, out1 => "Curvred Green Conv assembly")
   END_RUNG
   // the same network as SCL:
   IF "Green Lid Vision Sensor" THEN
       "Green lid Conv Assembly" := "ConvSpeedAfterMach";
       "Curvred Green Conv assembly" := "ConvSpeedAfterMach";
   END_IF;
   #_w1 := NOT "Green Lid Assembly Sensor" AND "Tag_5";   // falling edge of "Green Lid Assembly Sensor"
   "Tag_5" := "Green Lid Assembly Sensor";
   IF #_w1 OR "stop tag" THEN
       "Green lid Conv Assembly" := 0;
       "Curvred Green Conv assembly" := 0;
   END_IF;
END_REGION

REGION Network 31
   RUNG wire#powerrail
      P_Contact(operand := "Green Base Assembly Sensor", bit := "Tag_19")
      wire#w1
      I_Contact( "Tag_18" )
      Coil( "Clamp Green Base" )
   END_RUNG
   RUNG wire#powerrail
      Contact( "Clamp Green Base" )
   END_RUNG wire#w1
   // the same network as SCL:
   #_w1 := "Green Base Assembly Sensor" AND NOT "Tag_19";   // rising edge of "Green Base Assembly Sensor"
   "Tag_19" := "Green Base Assembly Sensor";
   "Clamp Green Base" := (#_w1 OR "Clamp Green Base") AND NOT "Tag_18";
END_REGION

REGION Network 32
   RUNG wire#powerrail
      P_Contact(operand := "Green Base Clamped", bit := "Tag_17")
      Coil( "Tag_18" )
   END_RUNG
   // the same network as SCL:
   #_w1 := "Green Base Clamped" AND NOT "Tag_17";   // rising edge of "Green Base Clamped"
   "Tag_17" := "Green Base Clamped";
   "Tag_18" := #_w1;
END_REGION

REGION Network 33
   RUNG wire#powerrail
      N_Contact(operand := "Green Lid Assembly Sensor", bit := "Tag_3")
      wire#w1
      I_Contact( "+ve edge to release G lid (true)" )
      Coil( "Clamp Green Lid" )
   END_RUNG
   RUNG wire#powerrail
      Contact( "Clamp Green Lid" )
   END_RUNG wire#w1
   RUNG wire#powerrail
      P_Contact(operand := "Green Lid Clamped", bit := "Tag_4")
      wire#w2
      Contact( "Clamp Green Lid" )
      Coil( "+ve edge to release G lid (true)" )
   END_RUNG
   RUNG wire#powerrail
      Contact( "+ve edge to release G lid (true)" )
   END_RUNG wire#w2
   // the same network as SCL:
   #_w1 := NOT "Green Lid Assembly Sensor" AND "Tag_3";   // falling edge of "Green Lid Assembly Sensor"
   "Tag_3" := "Green Lid Assembly Sensor";
   "Clamp Green Lid" := (#_w1 OR "Clamp Green Lid") AND NOT "+ve edge to release G lid (true)";
   #_w2 := "Green Lid Clamped" AND NOT "Tag_4";   // rising edge of "Green Lid Clamped"
   "Tag_4" := "Green Lid Clamped";
   "+ve edge to release G lid (true)" := (#_w2 OR "+ve edge to release G lid (true)") AND "Clamp Green Lid";
END_REGION

REGION Network 34
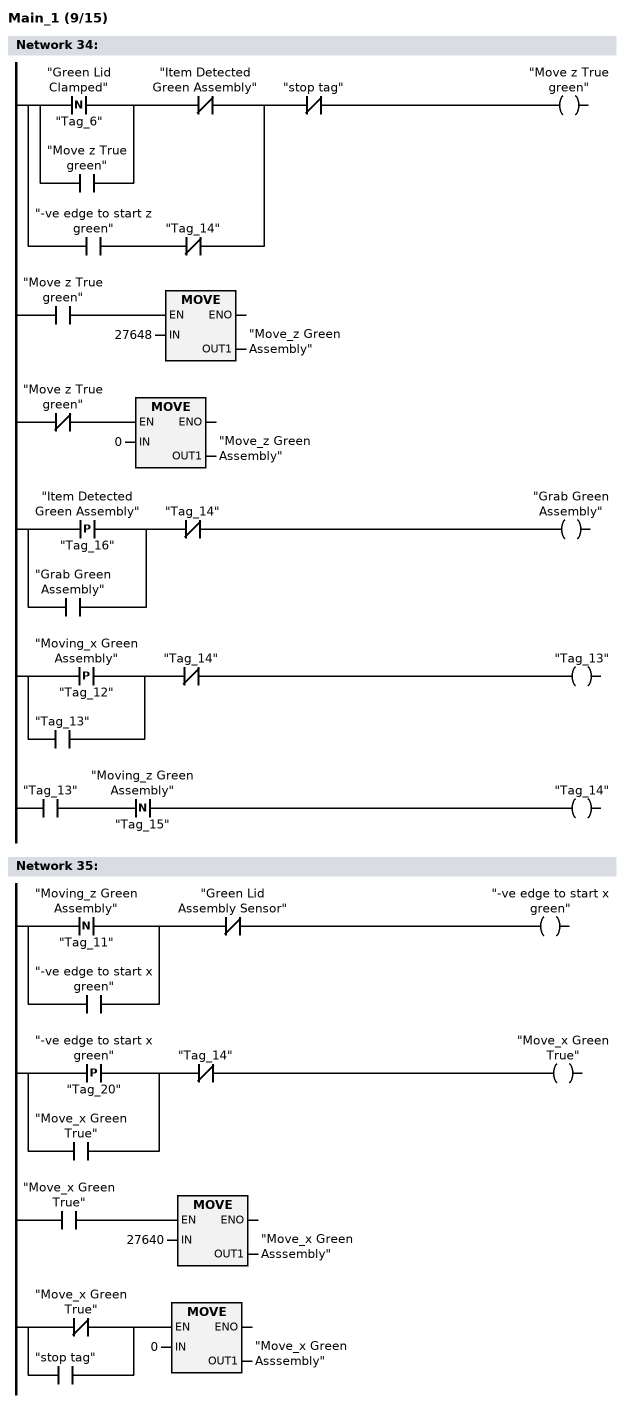
   RUNG wire#powerrail
      N_Contact(operand := "Green Lid Clamped", bit := "Tag_6")
      wire#w1
      I_Contact( "Item Detected Green Assembly" )
      wire#w2
      I_Contact( "stop tag" )
      Coil( "Move z True green" )
   END_RUNG
   RUNG wire#powerrail
      Contact( "Move z True green" )
   END_RUNG wire#w1
   RUNG wire#powerrail
      Contact( "-ve edge to start z green" )
      I_Contact( "Tag_14" )
   END_RUNG wire#w2
   RUNG wire#powerrail
      Contact( "Move z True green" )
      Move(in := 27648, out1 => "Move_z Green Assembly")
   END_RUNG
   RUNG wire#powerrail
      I_Contact( "Move z True green" )
      Move(in := 0, out1 => "Move_z Green Assembly")
   END_RUNG
   RUNG wire#powerrail
      P_Contact(operand := "Item Detected Green Assembly", bit := "Tag_16")
      wire#w3
      I_Contact( "Tag_14" )
      Coil( "Grab Green Assembly" )
   END_RUNG
   RUNG wire#powerrail
      Contact( "Grab Green Assembly" )
   END_RUNG wire#w3
   RUNG wire#powerrail
      P_Contact(operand := "Moving_x Green Assembly", bit := "Tag_12")
      wire#w4
      I_Contact( "Tag_14" )
      Coil( "Tag_13" )
   END_RUNG
   RUNG wire#powerrail
      Contact( "Tag_13" )
   END_RUNG wire#w4
   RUNG wire#powerrail
      Contact( "Tag_13" )
      N_Contact(operand := "Moving_z Green Assembly", bit := "Tag_15")
      Coil( "Tag_14" )
   END_RUNG
   // the same network as SCL:
   #_w1 := NOT "Green Lid Clamped" AND "Tag_6";   // falling edge of "Green Lid Clamped"
   "Tag_6" := "Green Lid Clamped";
   "Move z True green" := (((#_w1 OR "Move z True green") AND NOT "Item Detected Green Assembly") OR ("-ve edge to start z green" AND NOT "Tag_14")) AND NOT "stop tag";
   IF "Move z True green" THEN "Move_z Green Assembly" := 27648; END_IF;
   IF NOT "Move z True green" THEN "Move_z Green Assembly" := 0; END_IF;
   #_w2 := "Item Detected Green Assembly" AND NOT "Tag_16";   // rising edge of "Item Detected Green Assembly"
   "Tag_16" := "Item Detected Green Assembly";
   "Grab Green Assembly" := (#_w2 OR "Grab Green Assembly") AND NOT "Tag_14";
   #_w3 := "Moving_x Green Assembly" AND NOT "Tag_12";   // rising edge of "Moving_x Green Assembly"
   "Tag_12" := "Moving_x Green Assembly";
   "Tag_13" := (#_w3 OR "Tag_13") AND NOT "Tag_14";
   #_w4 := "Tag_13" AND NOT "Moving_z Green Assembly" AND "Tag_15";   // falling edge of "Moving_z Green Assembly"
   "Tag_15" := "Moving_z Green Assembly";
   "Tag_14" := #_w4;
END_REGION

REGION Network 35
   RUNG wire#powerrail
      N_Contact(operand := "Moving_z Green Assembly", bit := "Tag_11")
      wire#w1
      I_Contact( "Green Lid Assembly Sensor" )
      Coil( "-ve edge to start x green" )
   END_RUNG
   RUNG wire#powerrail
      Contact( "-ve edge to start x green" )
   END_RUNG wire#w1
   RUNG wire#powerrail
      P_Contact(operand := "-ve edge to start x green", bit := "Tag_20")
      wire#w2
      I_Contact( "Tag_14" )
      Coil( "Move_x Green True" )
   END_RUNG
   RUNG wire#powerrail
      Contact( "Move_x Green True" )
   END_RUNG wire#w2
   RUNG wire#powerrail
      Contact( "Move_x Green True" )
      Move(in := 27640, out1 => "Move_x Green Asssembly")
   END_RUNG
   RUNG wire#powerrail
      I_Contact( "Move_x Green True" )
      wire#w3
      Move(in := 0, out1 => "Move_x Green Asssembly")
   END_RUNG
   RUNG wire#powerrail
      Contact( "stop tag" )
   END_RUNG wire#w3
   // the same network as SCL:
   #_w1 := NOT "Moving_z Green Assembly" AND "Tag_11";   // falling edge of "Moving_z Green Assembly"
   "Tag_11" := "Moving_z Green Assembly";
   "-ve edge to start x green" := (#_w1 OR "-ve edge to start x green") AND NOT "Green Lid Assembly Sensor";
   #_w2 := "-ve edge to start x green" AND NOT "Tag_20";   // rising edge of "-ve edge to start x green"
   "Tag_20" := "-ve edge to start x green";
   "Move_x Green True" := (#_w2 OR "Move_x Green True") AND NOT "Tag_14";
   IF "Move_x Green True" THEN "Move_x Green Asssembly" := 27640; END_IF;
   IF NOT "Move_x Green True" OR "stop tag" THEN "Move_x Green Asssembly" := 0; END_IF;
END_REGION

REGION Network 36
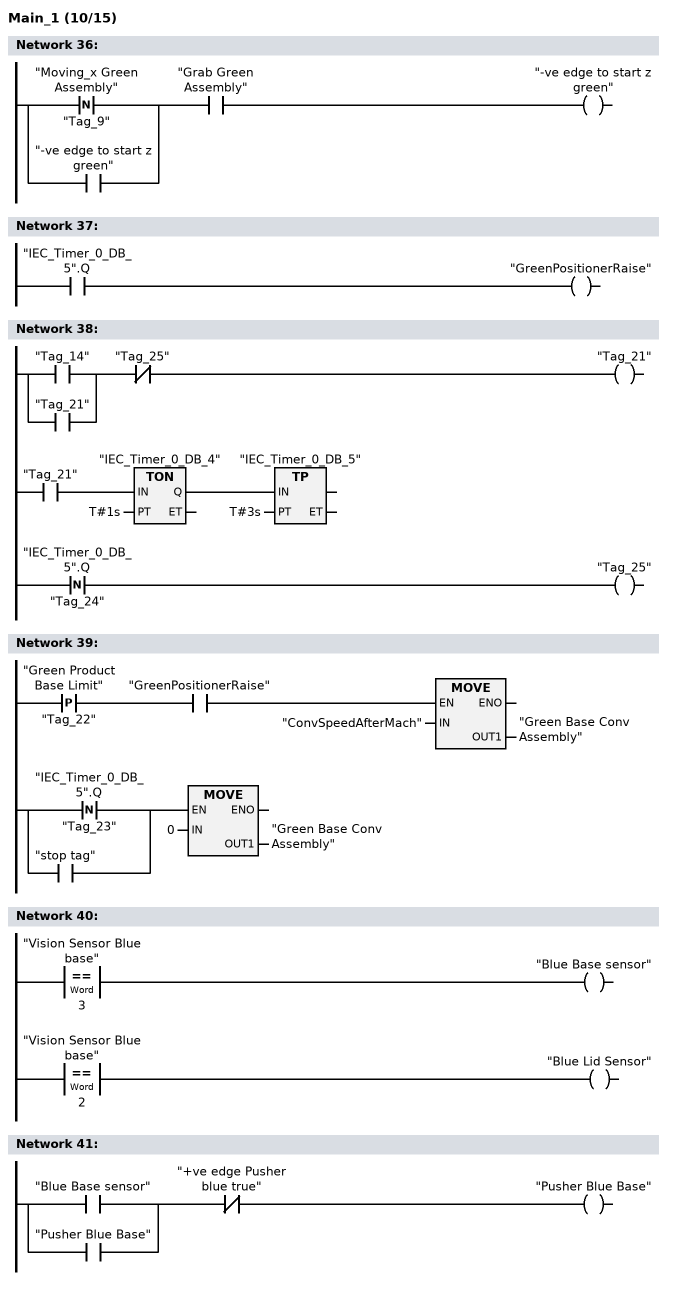
   RUNG wire#powerrail
      N_Contact(operand := "Moving_x Green Assembly", bit := "Tag_9")
      wire#w1
      Contact( "Grab Green Assembly" )
      Coil( "-ve edge to start z green" )
   END_RUNG
   RUNG wire#powerrail
      Contact( "-ve edge to start z green" )
   END_RUNG wire#w1
   // the same network as SCL:
   #_w1 := NOT "Moving_x Green Assembly" AND "Tag_9";   // falling edge of "Moving_x Green Assembly"
   "Tag_9" := "Moving_x Green Assembly";
   "-ve edge to start z green" := (#_w1 OR "-ve edge to start z green") AND "Grab Green Assembly";
END_REGION

REGION Network 37
   RUNG wire#powerrail
      Contact( "IEC_Timer_0_DB_5".Q )
      Coil( "GreenPositionerRaise" )
   END_RUNG
   // the same network as SCL:
   "GreenPositionerRaise" := "IEC_Timer_0_DB_5".Q;
END_REGION

REGION Network 38
   "Tag_21" := ("Tag_14" OR "Tag_21") AND NOT "Tag_25";
   "IEC_Timer_0_DB_4".TON(IN := "Tag_21", PT := T#1s);
   "IEC_Timer_0_DB_5".TP(IN := "IEC_Timer_0_DB_4".Q, PT := T#3s);
   #_w1 := NOT "IEC_Timer_0_DB_5".Q AND "Tag_24";   // falling edge of "IEC_Timer_0_DB_5".Q
   "Tag_24" := "IEC_Timer_0_DB_5".Q;
   "Tag_25" := #_w1;
END_REGION

REGION Network 39
   RUNG wire#powerrail
      P_Contact(operand := "Green Product Base Limit", bit := "Tag_22")
      Contact( "GreenPositionerRaise" )
      Move(in := "ConvSpeedAfterMach", out1 => "Green Base Conv Assembly")
   END_RUNG
   RUNG wire#powerrail
      N_Contact(operand := "IEC_Timer_0_DB_5".Q, bit := "Tag_23")
      wire#w1
      Move(in := 0, out1 => "Green Base Conv Assembly")
   END_RUNG
   RUNG wire#powerrail
      Contact( "stop tag" )
   END_RUNG wire#w1
   // the same network as SCL:
   #_w1 := "Green Product Base Limit" AND NOT "Tag_22";   // rising edge of "Green Product Base Limit"
   "Tag_22" := "Green Product Base Limit";
   IF #_w1 AND "GreenPositionerRaise" THEN "Green Base Conv Assembly" := "ConvSpeedAfterMach"; END_IF;
   #_w2 := NOT "IEC_Timer_0_DB_5".Q AND "Tag_23";   // falling edge of "IEC_Timer_0_DB_5".Q
   "Tag_23" := "IEC_Timer_0_DB_5".Q;
   IF #_w2 OR "stop tag" THEN "Green Base Conv Assembly" := 0; END_IF;
END_REGION

REGION Network 40
   RUNG wire#powerrail
      { S7_Templates := "SrcType := Word" } EQ_Contact(in1 := "Vision Sensor Blue base", in2 := 3)
      Coil( "Blue Base sensor" )
   END_RUNG
   RUNG wire#powerrail
      { S7_Templates := "SrcType := Word" } EQ_Contact(in1 := "Vision Sensor Blue base", in2 := 2)
      Coil( "Blue Lid Sensor" )
   END_RUNG
   // the same network as SCL:
   "Blue Base sensor" := "Vision Sensor Blue base" = 3;
   "Blue Lid Sensor" := "Vision Sensor Blue base" = 2;
END_REGION

REGION Network 41
   RUNG wire#powerrail
      Contact( "Blue Base sensor" )
      wire#w1
      I_Contact( "+ve edge Pusher blue true" )
      Coil( "Pusher Blue Base" )
   END_RUNG
   RUNG wire#powerrail
      Contact( "Pusher Blue Base" )
   END_RUNG wire#w1
   // the same network as SCL:
   "Pusher Blue Base" := ("Blue Base sensor" OR "Pusher Blue Base") AND NOT "+ve edge Pusher blue true";
END_REGION

REGION Network 42
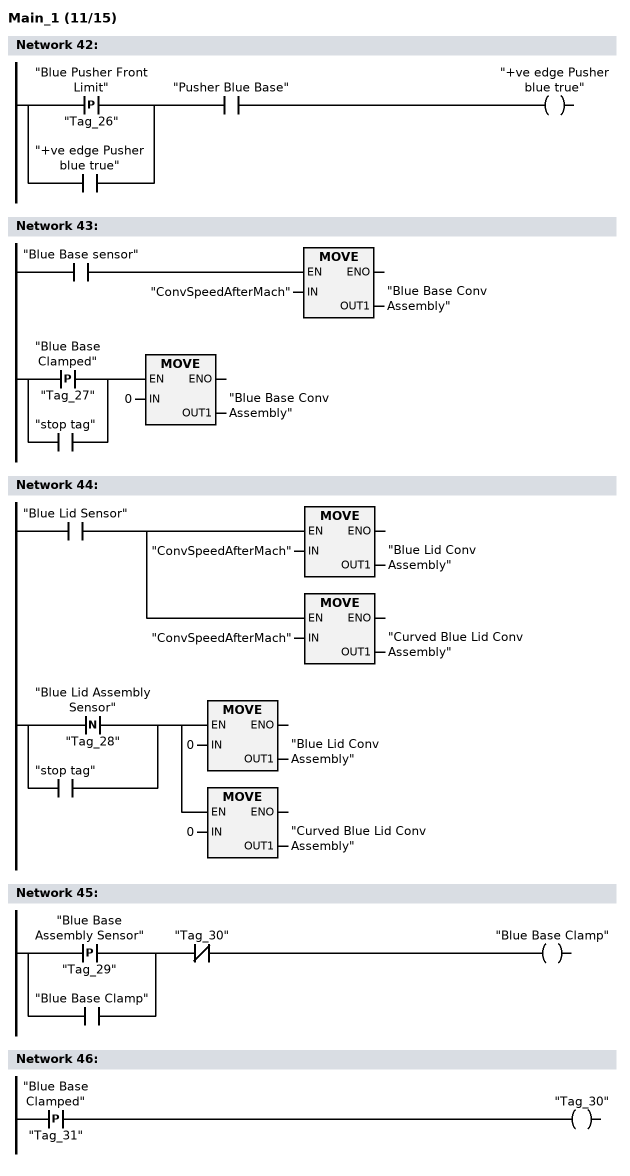
   RUNG wire#powerrail
      P_Contact(operand := "Blue Pusher Front Limit", bit := "Tag_26")
      wire#w1
      Contact( "Pusher Blue Base" )
      Coil( "+ve edge Pusher blue true" )
   END_RUNG
   RUNG wire#powerrail
      Contact( "+ve edge Pusher blue true" )
   END_RUNG wire#w1
   // the same network as SCL:
   #_w1 := "Blue Pusher Front Limit" AND NOT "Tag_26";   // rising edge of "Blue Pusher Front Limit"
   "Tag_26" := "Blue Pusher Front Limit";
   "+ve edge Pusher blue true" := (#_w1 OR "+ve edge Pusher blue true") AND "Pusher Blue Base";
END_REGION

REGION Network 43
   RUNG wire#powerrail
      Contact( "Blue Base sensor" )
      Move(in := "ConvSpeedAfterMach", out1 => "Blue Base Conv Assembly")
   END_RUNG
   RUNG wire#powerrail
      P_Contact(operand := "Blue Base Clamped", bit := "Tag_27")
      wire#w1
      Move(in := 0, out1 => "Blue Base Conv Assembly")
   END_RUNG
   RUNG wire#powerrail
      Contact( "stop tag" )
   END_RUNG wire#w1
   // the same network as SCL:
   IF "Blue Base sensor" THEN "Blue Base Conv Assembly" := "ConvSpeedAfterMach"; END_IF;
   #_w1 := "Blue Base Clamped" AND NOT "Tag_27";   // rising edge of "Blue Base Clamped"
   "Tag_27" := "Blue Base Clamped";
   IF #_w1 OR "stop tag" THEN "Blue Base Conv Assembly" := 0; END_IF;
END_REGION

REGION Network 44
   RUNG wire#powerrail
      Contact( "Blue Lid Sensor" )
      wire#w1
      Move(in := "ConvSpeedAfterMach", out1 => "Blue Lid Conv Assembly")
   END_RUNG
   RUNG wire#w1
      Move(in := "ConvSpeedAfterMach", out1 => "Curved Blue Lid Conv Assembly")
   END_RUNG
   RUNG wire#powerrail
      N_Contact(operand := "Blue Lid Assembly Sensor", bit := "Tag_28")
      wire#w2
      Move(in := 0, out1 => "Blue Lid Conv Assembly")
   END_RUNG
   RUNG wire#powerrail
      Contact( "stop tag" )
   END_RUNG wire#w2
   RUNG wire#w2
      Move(in := 0, out1 => "Curved Blue Lid Conv Assembly")
   END_RUNG
   // the same network as SCL:
   IF "Blue Lid Sensor" THEN
       "Blue Lid Conv Assembly" := "ConvSpeedAfterMach";
       "Curved Blue Lid Conv Assembly" := "ConvSpeedAfterMach";
   END_IF;
   #_w1 := NOT "Blue Lid Assembly Sensor" AND "Tag_28";   // falling edge of "Blue Lid Assembly Sensor"
   "Tag_28" := "Blue Lid Assembly Sensor";
   IF #_w1 OR "stop tag" THEN
       "Blue Lid Conv Assembly" := 0;
       "Curved Blue Lid Conv Assembly" := 0;
   END_IF;
END_REGION

REGION Network 45
   RUNG wire#powerrail
      P_Contact(operand := "Blue Base Assembly Sensor", bit := "Tag_29")
      wire#w1
      I_Contact( "Tag_30" )
      Coil( "Blue Base Clamp" )
   END_RUNG
   RUNG wire#powerrail
      Contact( "Blue Base Clamp" )
   END_RUNG wire#w1
   // the same network as SCL:
   #_w1 := "Blue Base Assembly Sensor" AND NOT "Tag_29";   // rising edge of "Blue Base Assembly Sensor"
   "Tag_29" := "Blue Base Assembly Sensor";
   "Blue Base Clamp" := (#_w1 OR "Blue Base Clamp") AND NOT "Tag_30";
END_REGION

REGION Network 46
   RUNG wire#powerrail
      P_Contact(operand := "Blue Base Clamped", bit := "Tag_31")
      Coil( "Tag_30" )
   END_RUNG
   // the same network as SCL:
   #_w1 := "Blue Base Clamped" AND NOT "Tag_31";   // rising edge of "Blue Base Clamped"
   "Tag_31" := "Blue Base Clamped";
   "Tag_30" := #_w1;
END_REGION

REGION Network 47
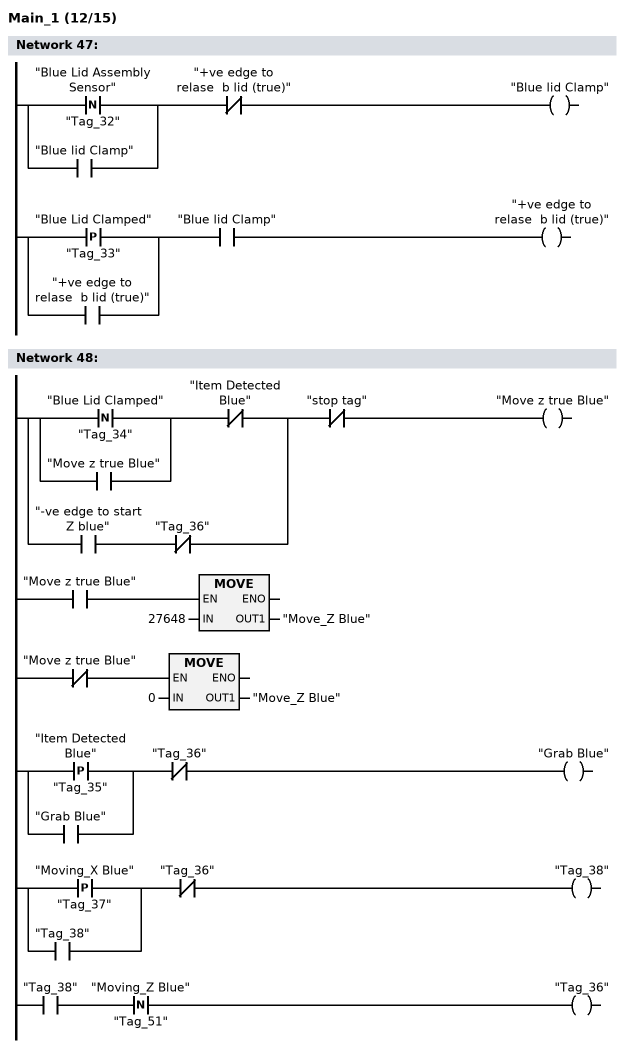
   RUNG wire#powerrail
      N_Contact(operand := "Blue Lid Assembly Sensor", bit := "Tag_32")
      wire#w1
      I_Contact( "+ve edge to relase  b lid (true)" )
      Coil( "Blue lid Clamp" )
   END_RUNG
   RUNG wire#powerrail
      Contact( "Blue lid Clamp" )
   END_RUNG wire#w1
   RUNG wire#powerrail
      P_Contact(operand := "Blue Lid Clamped", bit := "Tag_33")
      wire#w2
      Contact( "Blue lid Clamp" )
      Coil( "+ve edge to relase  b lid (true)" )
   END_RUNG
   RUNG wire#powerrail
      Contact( "+ve edge to relase  b lid (true)" )
   END_RUNG wire#w2
   // the same network as SCL:
   #_w1 := NOT "Blue Lid Assembly Sensor" AND "Tag_32";   // falling edge of "Blue Lid Assembly Sensor"
   "Tag_32" := "Blue Lid Assembly Sensor";
   "Blue lid Clamp" := (#_w1 OR "Blue lid Clamp") AND NOT "+ve edge to relase  b lid (true)";
   #_w2 := "Blue Lid Clamped" AND NOT "Tag_33";   // rising edge of "Blue Lid Clamped"
   "Tag_33" := "Blue Lid Clamped";
   "+ve edge to relase  b lid (true)" := (#_w2 OR "+ve edge to relase  b lid (true)") AND "Blue lid Clamp";
END_REGION

REGION Network 48
   RUNG wire#powerrail
      N_Contact(operand := "Blue Lid Clamped", bit := "Tag_34")
      wire#w1
      I_Contact( "Item Detected Blue" )
      wire#w2
      I_Contact( "stop tag" )
      Coil( "Move z true Blue" )
   END_RUNG
   RUNG wire#powerrail
      Contact( "Move z true Blue" )
   END_RUNG wire#w1
   RUNG wire#powerrail
      Contact( "-ve edge to start Z blue" )
      I_Contact( "Tag_36" )
   END_RUNG wire#w2
   RUNG wire#powerrail
      Contact( "Move z true Blue" )
      Move(in := 27648, out1 => "Move_Z Blue")
   END_RUNG
   RUNG wire#powerrail
      I_Contact( "Move z true Blue" )
      Move(in := 0, out1 => "Move_Z Blue")
   END_RUNG
   RUNG wire#powerrail
      P_Contact(operand := "Item Detected Blue", bit := "Tag_35")
      wire#w3
      I_Contact( "Tag_36" )
      Coil( "Grab Blue" )
   END_RUNG
   RUNG wire#powerrail
      Contact( "Grab Blue" )
   END_RUNG wire#w3
   RUNG wire#powerrail
      P_Contact(operand := "Moving_X Blue", bit := "Tag_37")
      wire#w4
      I_Contact( "Tag_36" )
      Coil( "Tag_38" )
   END_RUNG
   RUNG wire#powerrail
      Contact( "Tag_38" )
   END_RUNG wire#w4
   RUNG wire#powerrail
      Contact( "Tag_38" )
      N_Contact(operand := "Moving_Z Blue", bit := "Tag_51")
      Coil( "Tag_36" )
   END_RUNG
   // the same network as SCL:
   #_w1 := NOT "Blue Lid Clamped" AND "Tag_34";   // falling edge of "Blue Lid Clamped"
   "Tag_34" := "Blue Lid Clamped";
   "Move z true Blue" := (((#_w1 OR "Move z true Blue") AND NOT "Item Detected Blue") OR ("-ve edge to start Z blue" AND NOT "Tag_36")) AND NOT "stop tag";
   IF "Move z true Blue" THEN "Move_Z Blue" := 27648; END_IF;
   IF NOT "Move z true Blue" THEN "Move_Z Blue" := 0; END_IF;
   #_w2 := "Item Detected Blue" AND NOT "Tag_35";   // rising edge of "Item Detected Blue"
   "Tag_35" := "Item Detected Blue";
   "Grab Blue" := (#_w2 OR "Grab Blue") AND NOT "Tag_36";
   #_w3 := "Moving_X Blue" AND NOT "Tag_37";   // rising edge of "Moving_X Blue"
   "Tag_37" := "Moving_X Blue";
   "Tag_38" := (#_w3 OR "Tag_38") AND NOT "Tag_36";
   #_w4 := "Tag_38" AND NOT "Moving_Z Blue" AND "Tag_51";   // falling edge of "Moving_Z Blue"
   "Tag_51" := "Moving_Z Blue";
   "Tag_36" := #_w4;
END_REGION

REGION Network 49
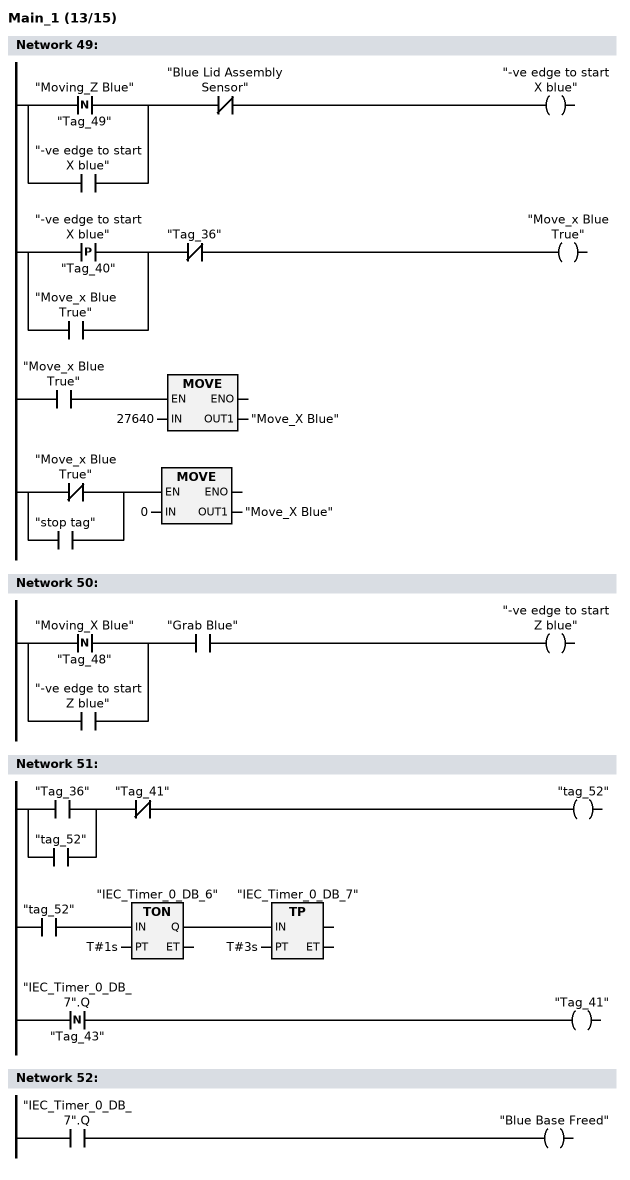
   RUNG wire#powerrail
      N_Contact(operand := "Moving_Z Blue", bit := "Tag_49")
      wire#w1
      I_Contact( "Blue Lid Assembly Sensor" )
      Coil( "-ve edge to start X blue" )
   END_RUNG
   RUNG wire#powerrail
      Contact( "-ve edge to start X blue" )
   END_RUNG wire#w1
   RUNG wire#powerrail
      P_Contact(operand := "-ve edge to start X blue", bit := "Tag_40")
      wire#w2
      I_Contact( "Tag_36" )
      Coil( "Move_x Blue True" )
   END_RUNG
   RUNG wire#powerrail
      Contact( "Move_x Blue True" )
   END_RUNG wire#w2
   RUNG wire#powerrail
      Contact( "Move_x Blue True" )
      Move(in := 27640, out1 => "Move_X Blue")
   END_RUNG
   RUNG wire#powerrail
      I_Contact( "Move_x Blue True" )
      wire#w3
      Move(in := 0, out1 => "Move_X Blue")
   END_RUNG
   RUNG wire#powerrail
      Contact( "stop tag" )
   END_RUNG wire#w3
   // the same network as SCL:
   #_w1 := NOT "Moving_Z Blue" AND "Tag_49";   // falling edge of "Moving_Z Blue"
   "Tag_49" := "Moving_Z Blue";
   "-ve edge to start X blue" := (#_w1 OR "-ve edge to start X blue") AND NOT "Blue Lid Assembly Sensor";
   #_w2 := "-ve edge to start X blue" AND NOT "Tag_40";   // rising edge of "-ve edge to start X blue"
   "Tag_40" := "-ve edge to start X blue";
   "Move_x Blue True" := (#_w2 OR "Move_x Blue True") AND NOT "Tag_36";
   IF "Move_x Blue True" THEN "Move_X Blue" := 27640; END_IF;
   IF NOT "Move_x Blue True" OR "stop tag" THEN "Move_X Blue" := 0; END_IF;
END_REGION

REGION Network 50
   RUNG wire#powerrail
      N_Contact(operand := "Moving_X Blue", bit := "Tag_48")
      wire#w1
      Contact( "Grab Blue" )
      Coil( "-ve edge to start Z blue" )
   END_RUNG
   RUNG wire#powerrail
      Contact( "-ve edge to start Z blue" )
   END_RUNG wire#w1
   // the same network as SCL:
   #_w1 := NOT "Moving_X Blue" AND "Tag_48";   // falling edge of "Moving_X Blue"
   "Tag_48" := "Moving_X Blue";
   "-ve edge to start Z blue" := (#_w1 OR "-ve edge to start Z blue") AND "Grab Blue";
END_REGION

REGION Network 51
   "tag_52" := ("Tag_36" OR "tag_52") AND NOT "Tag_41";
   "IEC_Timer_0_DB_6".TON(IN := "tag_52", PT := T#1s);
   "IEC_Timer_0_DB_7".TP(IN := "IEC_Timer_0_DB_6".Q, PT := T#3s);
   #_w1 := NOT "IEC_Timer_0_DB_7".Q AND "Tag_43";   // falling edge of "IEC_Timer_0_DB_7".Q
   "Tag_43" := "IEC_Timer_0_DB_7".Q;
   "Tag_41" := #_w1;
END_REGION

REGION Network 52
   RUNG wire#powerrail
      Contact( "IEC_Timer_0_DB_7".Q )
      Coil( "Blue Base Freed" )
   END_RUNG
   // the same network as SCL:
   "Blue Base Freed" := "IEC_Timer_0_DB_7".Q;
END_REGION

REGION Network 53
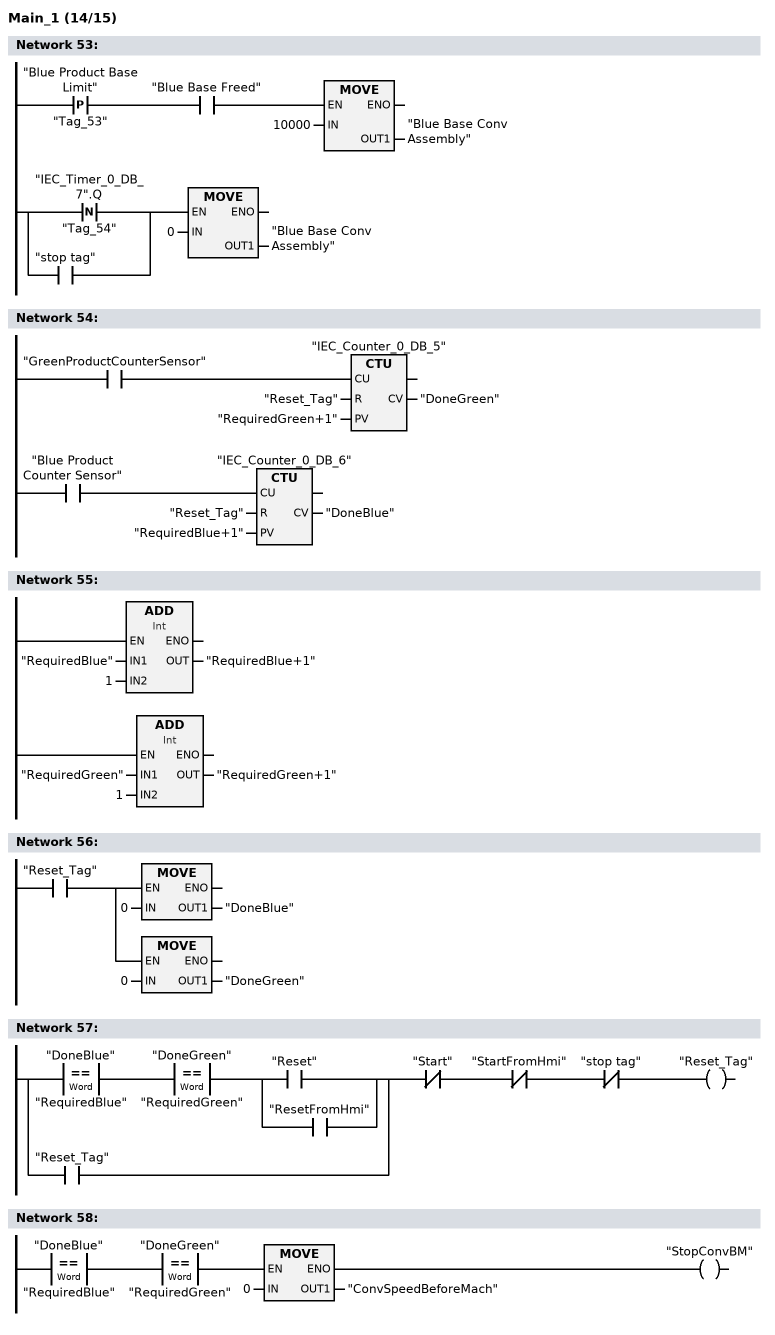
   RUNG wire#powerrail
      P_Contact(operand := "Blue Product Base Limit", bit := "Tag_53")
      Contact( "Blue Base Freed" )
      Move(in := 10000, out1 => "Blue Base Conv Assembly")
   END_RUNG
   RUNG wire#powerrail
      N_Contact(operand := "IEC_Timer_0_DB_7".Q, bit := "Tag_54")
      wire#w1
      Move(in := 0, out1 => "Blue Base Conv Assembly")
   END_RUNG
   RUNG wire#powerrail
      Contact( "stop tag" )
   END_RUNG wire#w1
   // the same network as SCL:
   #_w1 := "Blue Product Base Limit" AND NOT "Tag_53";   // rising edge of "Blue Product Base Limit"
   "Tag_53" := "Blue Product Base Limit";
   IF #_w1 AND "Blue Base Freed" THEN "Blue Base Conv Assembly" := 10000; END_IF;
   #_w2 := NOT "IEC_Timer_0_DB_7".Q AND "Tag_54";   // falling edge of "IEC_Timer_0_DB_7".Q
   "Tag_54" := "IEC_Timer_0_DB_7".Q;
   IF #_w2 OR "stop tag" THEN "Blue Base Conv Assembly" := 0; END_IF;
END_REGION

REGION Network 54
   "IEC_Counter_0_DB_5".CTU(CU := "GreenProductCounterSensor",
                           R := "Reset_Tag",
                           PV := "RequiredGreen+1",
                           CV => "DoneGreen");
   "IEC_Counter_0_DB_6".CTU(CU := "Blue Product Counter Sensor",
                           R := "Reset_Tag",
                           PV := "RequiredBlue+1",
                           CV => "DoneBlue");
END_REGION

REGION Network 55
   RUNG wire#powerrail
      { S7_Templates := "SrcType := Int" } Add(in1 := "RequiredBlue", in2 := 1, out => "RequiredBlue+1")
   END_RUNG
   RUNG wire#powerrail
      { S7_Templates := "SrcType := Int" } Add(in1 := "RequiredGreen", in2 := 1, out => "RequiredGreen+1")
   END_RUNG
   // the same network as SCL:
   "RequiredBlue+1" := "RequiredBlue" + 1;
   "RequiredGreen+1" := "RequiredGreen" + 1;
END_REGION

REGION Network 56
   RUNG wire#powerrail
      Contact( "Reset_Tag" )
      wire#w1
      Move(in := 0, out1 => "DoneBlue")
   END_RUNG
   RUNG wire#w1
      Move(in := 0, out1 => "DoneGreen")
   END_RUNG
   // the same network as SCL:
   IF "Reset_Tag" THEN
       "DoneBlue" := 0;
       "DoneGreen" := 0;
   END_IF;
END_REGION

REGION Network 57
   RUNG wire#powerrail
      { S7_Templates := "SrcType := Word" } EQ_Contact(in1 := "DoneBlue", in2 := "RequiredBlue")
      { S7_Templates := "SrcType := Word" } EQ_Contact(in1 := "DoneGreen", in2 := "RequiredGreen")
      wire#w1
      Contact( "Reset" )
      wire#w2
      I_Contact( "Start" )
      I_Contact( "StartFromHmi" )
      I_Contact( "stop tag" )
      Coil( "Reset_Tag" )
   END_RUNG
   RUNG wire#w1
      Contact( "ResetFromHmi" )
   END_RUNG wire#w2
   RUNG wire#powerrail
      Contact( "Reset_Tag" )
   END_RUNG wire#w2
   // the same network as SCL:
   "Reset_Tag" := ((("DoneBlue" = "RequiredBlue") AND ("DoneGreen" = "RequiredGreen") AND ("Reset" OR "ResetFromHmi")) OR "Reset_Tag") AND NOT "Start" AND NOT "StartFromHmi" AND NOT "stop tag";
END_REGION

REGION Network 58
   RUNG wire#powerrail
      { S7_Templates := "SrcType := Word" } EQ_Contact(in1 := "DoneBlue", in2 := "RequiredBlue")
      { S7_Templates := "SrcType := Word" } EQ_Contact(in1 := "DoneGreen", in2 := "RequiredGreen")
      Move(in := 0, out1 => "ConvSpeedBeforeMach")
      Coil( "StopConvBM" )
   END_RUNG
   // the same network as SCL:
   #_w1 := ("DoneBlue" = "RequiredBlue") AND ("DoneGreen" = "RequiredGreen");
   IF #_w1 THEN "ConvSpeedBeforeMach" := 0; END_IF;
   "StopConvBM" := #_w1;
END_REGION

REGION Network 59
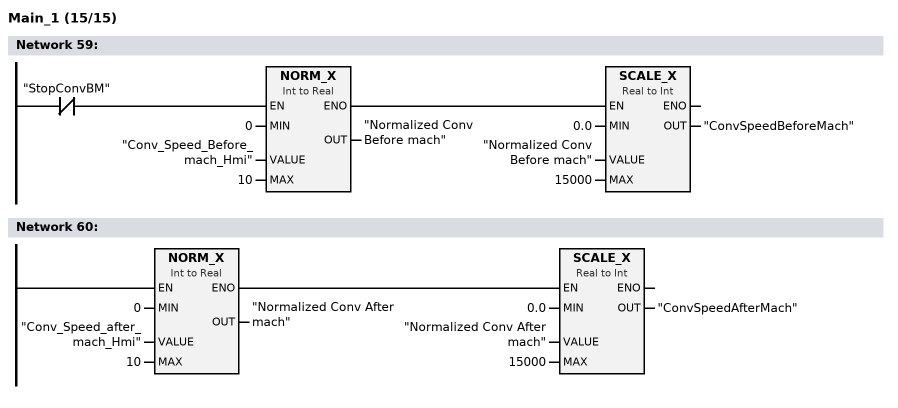
   RUNG wire#powerrail
      I_Contact( "StopConvBM" )
      { S7_Templates := "[SrcType := Int, DestType := Real]" } Normalize(min := 0, value := "Conv_Speed_Before_mach_Hmi", max := 10, out => "Normalized Conv Before mach")
      { S7_Templates := "[SrcType := Real, DestType := Int]" } Scale(min := 0.0, value := "Normalized Conv Before mach", max := 15000, out => "ConvSpeedBeforeMach")
   END_RUNG
   // the same network as SCL:
   IF NOT "StopConvBM" THEN
       "Normalized Conv Before mach" := NORM_X(MIN := 0, VALUE := "Conv_Speed_Before_mach_Hmi", MAX := 10);
       "ConvSpeedBeforeMach" := SCALE_X(MIN := 0.0, VALUE := "Normalized Conv Before mach", MAX := 15000);
   END_IF;
END_REGION

REGION Network 60
   RUNG wire#powerrail
      { S7_Templates := "[SrcType := Int, DestType := Real]" } Normalize(min := 0, value := "Conv_Speed_after_mach_Hmi", max := 10, out => "Normalized Conv After mach")
      { S7_Templates := "[SrcType := Real, DestType := Int]" } Scale(min := 0.0, value := "Normalized Conv After mach", max := 15000, out => "ConvSpeedAfterMach")
   END_RUNG
   // the same network as SCL:
   "Normalized Conv After mach" := NORM_X(MIN := 0, VALUE := "Conv_Speed_after_mach_Hmi", MAX := 10);
   "ConvSpeedAfterMach" := SCALE_X(MIN := 0.0, VALUE := "Normalized Conv After mach", MAX := 15000);
END_REGION
END_ORGANIZATION_BLOCK

(* ===== HMI "HMI_RT_2" =====
system functions are stored by id; their names below are inferred from use
connection "HMI_Connection_2": ETHERNET, S7_1500_OMS

HMI tags "Default tag table"
   "Tag_ScreenNumber" : UInt, internal
   "DoneBlue" : Word = PLC DoneBlue AT %MW710, 1 s
   "DoneGreen" : Word = PLC DoneGreen AT %MW708, 1 s
   "RequiredBlue" : Word = PLC RequiredBlue AT %MW702, 1 s
   "RequiredGreen" : Word = PLC RequiredGreen AT %MW700, 1 s
   "StartFromHMI" : Bool = PLC StartFromHmi AT %M601.4, 1 s
   "Start Light" : Bool = PLC "Start Light" AT %Q0.5, 1 s
   "ConvSpeedBeforeMach(1)" : Word = PLC Conv_Speed_Before_mach_Hmi AT %MW724
   "ConvSpeedAfterMach(1)" : Word = PLC Conv_Speed_after_mach_Hmi AT %MW726, 1 s
   "StopFromHmi" : Bool = PLC StopFromHmi AT %M601.5, 1 s
   "ResetFromHmi" : Bool = PLC ResetFromHmi AT %M601.6, 1 s
   "Stop Light" : Bool = PLC "Stop Light" AT %Q0.7, 1 s
   "Reset Light" : Bool = PLC "Reset Light" AT %Q0.6, 1 s

screen "Control and DAQ" 1280x740, template "Template_1"
   on GenerateScreen: SetTag("Tag_ScreenNumber", 1)
   GraphicView "Graphic view_1" at 0,4 size 1276x736; Picture "COVER HMI"
   Slider "Slider_1" at 300,144 size 80x230; Caption 'V'
      ProcessValue <- "ConvSpeedBeforeMach(1)"
   TextField "HmiScreenItemData_1" at 184,30 size 1024x65; Text 'Welcome to Our Factory'
   IOField "I/O field_1" at 157,475 size 96x32; FormatPattern 99
      ProcessValue <- "RequiredBlue"
   IOField "I/O field_2" at 467,473 size 96x32; FormatPattern 99
      ProcessValue <- "RequiredGreen"
   IOField "I/O field_3" at 814,470 size 96x32; FormatPattern 99
      ProcessValue <- "DoneBlue"
   IOField "I/O field_4" at 1090,474 size 96x32; FormatPattern 99
      ProcessValue <- "DoneGreen"
   TextField "Text field_1" at 126,423 size 229x46; Text 'Required Number Of Blue Products'
   TextField "Text field_2" at 406,423 size 221x46; Text 'Required Number of Green Products'
   TextField "Text field_3" at 751,414 size 216x46; Text 'Assembled Blue Products'
   TextField "Text field_4" at 1030,423 size 224x46; Text 'Assembled Green Products'
   TextField "Text field_5" at 147,114 size 373x25; Text 'Conveyor Speed Before machining'
   TextField "Text field_6" at 767,111 size 357x25; Text 'Conveyor Speed After Machining'
   Slider "Slider_2" at 887,147 size 80x230; Caption 'V'
      ProcessValue <- "ConvSpeedAfterMach(1)"
   Button "Button_4" at 267,630 size 96x32; TextOff 'Start'
      on Press: function_b14e0dd5("StartFromHMI", 0)
   Circle "Circle_4" at 284,555 size 63x63
      Appearance <- "Start Light"
   Button "Button_5" at 575,630 size 96x32; TextOff 'Stop'
      on Press: function_b14e0dd5("StopFromHmi", 0)
   Circle "Circle_5" at 592,555 size 63x63
      Appearance <- "Stop Light"
   Button "Button_6" at 845,628 size 96x32; TextOff 'Reset'
      on Press: function_b14e0dd5("ResetFromHmi", 0)
   Circle "Circle_6" at 862,553 size 63x63
      Appearance <- "Reset Light"

Template "Template_1" 1280x740
   Button "Exit" at 1200,679 size 78x59; TextOff 'Exit'; PictureOff "ExitRuntime_TP1200_Comfort_TR"; PictureOn "ExitRuntime_TP1200_Comfort_TR"
      on Release: StopRuntime(0)
   Button "Template_Button" at 1120,679 size 78x59; TextOff 'Text'
   Button "Template_Button_1" at 1040,679 size 78x59; TextOff 'Text'
   Button "Template_Button_2" at 960,679 size 78x59; TextOff 'Text'
   Button "Template_Button_3" at 880,679 size 78x59; TextOff 'Text'
   Button "Template_Button_4" at 800,679 size 78x59; TextOff 'Text'
   Button "Template_Button_5" at 720,679 size 78x59; TextOff 'Text'
   Button "Template_Button_6" at 640,679 size 78x59; TextOff 'Text'
   Button "Template_Button_7" at 561,679 size 78x59; TextOff 'Text'
   Button "Template_Button_8" at 481,679 size 78x59; TextOff 'Text'
   Button "Template_Button_9" at 401,679 size 78x59; TextOff 'Text'
   Button "Template_Button_10" at 321,679 size 78x59; TextOff 'Text'
   Button "Template_Button_11" at 241,679 size 78x59; TextOff 'Text'
   Button "Template_Button_12" at 161,679 size 78x59; TextOff 'Text'
   Button "Alarms" at 81,679 size 78x59; TextOff 'Alarms'; PictureOff "AlarmDisplay_TP1200_Comfort_TR"; PictureOn "AlarmDisplay_TP1200_Comfort_TR"
      on Release: function_ef3f5d25("Alarm window_Unacknowledged", -1)
   Button "Start screen" at 1,679 size 78x59; TextOff 'Start screen'; PictureOff "NavigateHome_TP1200_Comfort_TR"; PictureOn "NavigateHome_TP1200_Comfort_TR"
      on Release: ActivateScreen("Control and DAQ", 0)
*)